// TIA Portal V19 export
FUNCTION_BLOCK "HMI_A03_FB"   // FB63, LAD
TITLE = HMI Managment
AUTHOR : Piemme
FAMILY : System
// stored: MemoryReserve 100, SetENOAutomatically false
   VAR_OUTPUT
      MB3_LpJog : Bool;
   END_VAR
   VAR
      MB3_Decoder { ExternalAccessible := 'False'; ExternalVisible := 'False'; ExternalWritable := 'False'} : "ButtonsHMIDecoder";
   END_VAR
   VAR CONSTANT
      "3002_TRASPORTO" : Int := 3002;
      "3011_FERMI_P1" : Int := 3011;
      "3012_FERMI_P1_SFALSATORE" : Int := 3012;
      "3021_FERMI_P2" : Int := 3021;
      "3022_FERMI_P2_SOLLEVATORE" : Int := 3022;
      "3031_FERMI_P3" : Int := 3031;
      "3032_SOLLEVA_RIBALTA" : Int := 3032;
      "3033_ROT_RIBALTA" : Int := 3033;
      "3034_ROT_RIBALTA_AX-POS" : Int := 3034;
      "3041_FERMI_P4" : Int := 3041;
      "3042_SPINTORE_LAT_VRT_P5" : Int := 3042;
      "3043_SPINTORE_LAT_ORZ_P5" : Int := 3043;
      "3044_SOLLEVATORI_P5" : Int := 3044;
      "3045_SPINTORE_LAT_OP" : Int := 3045;
      "3051_RIBALTATORE_OP-POS0" : Int := 3051;
      "3052_RIBALTATORE_OP-POS1" : Int := 3052;
      "3053_RIBALTATORE_OP-POS2" : Int := 3053;
      "3054_RIBALTATORE_OP-POS3" : Int := 3054;
      "4001_HU_CYTROPACK" : Int := 4001;
      "4011_SPINTORE_OP" : Int := 4011;
      "4012_SPINTORE_AX" : Int := 4012;
      "4013_SPINTORE_VRT" : Int := 4013;
      "4014_SPINTORE_ORZ" : Int := 4014;
      "4021_BORDATRICE_AX" : Int := 4021;
      "4031_RULLIERA_OP" : Int := 4031;
      "4032_RULLIERA_AX" : Int := 4032;
      "4033_BORDATRICE_REG-CASSETTA" : Int := 4033;
      "4034_BORDATRICE_PASS01" : Int := 4034;
      "4035_BORDATRICE_PASS02" : Int := 4035;
      "4036_BORDATRICE_PASS03" : Int := 4036;
      "4037_BORDATRICE_PASS04" : Int := 4037;
      "4038_BORDATRICE_REG-CASSETTA_AX-POS" : Int := 4038;
      "4041_CENTRATORI_OP" : Int := 4041;
      "4042_CENTRATORI_CENTRAGGIO" : Int := 4042;
      "4043_CENTRATORI_SOLLEVAMENTO" : Int := 4043;
      "4051_PAREGGIATORE_CODA_OP" : Int := 4051;
      "4052_PAREGGIATORE_CODA_AX" : Int := 4052;
      "4053_PAREGGIATORE_CODA_BLOCCAGGIO" : Int := 4053;
      "4054_PAREGGIATORE_CODA_BATTUTAVERTICALE" : Int := 4054;
      "4055_PAREGGIATORE_CODA_PAREGGIATORELONGIT" : Int := 4055;
      "4061_PAREGGIATORE_TESTA_OP" : Int := 4061;
      "4062_PAREGGIATORE_TESTA_AX" : Int := 4062;
      "4063_PAREGGIATORE_TESTA_BLOCCAGGIO" : Int := 4063;
      "4064_PAREGGIATORE_TESTA_SOLLEVAMENTO" : Int := 4064;
      "4065_PAREGGIATORE_TESTA_CENTRAGGIO" : Int := 4065;
      "4066_PAREGG_TESTA_AX_POS" : Int := 4066;
      "4067_PAREGG_CODA_AX_POS" : Int := 4067;
      "4070_MANIPOLATORE_OP" : Int := 4070;
      "4071_MANIPOLATORE_AX" : Int := 4071;
      "4072_MANIPOLATORE_AX-POS" : Int := 4072;
      "4073_MANIPOLATORE_MAGNETE" : Int := 4073;
      "4074_MANIPOLATORE_SOLLEVATORE" : Int := 4074;
      "4080_BORDATRICE_PASS01_LATO-OP" : Int := 4080;
      "4081_BORDATRICE_PASS01_LATO-MOT" : Int := 4081;
      "4082_BORDATRICE_PASS02_LATO-OP" : Int := 4082;
      "4083_BORDATRICE_PASS02_LATO-MOT" : Int := 4083;
      "4084_BORDATRICE_PASS03_LATO-OP" : Int := 4084;
      "4085_BORDATRICE_PASS03_LATO-MOT" : Int := 4085;
      "4086_BORDATRICE_PASS04_LATO-OP" : Int := 4086;
      "4087_BORDATRICE_PASS04_LATO-MOT" : Int := 4087;
      "4088_BORDATRICE_PASS01-COMBO_AX-POS" : Int := 4088;
      "4089_BORDATRICE_PASS02-COMBO_AX-POS" : Int := 4089;
      "4090_BORDATRICE_PASS03-COMBO_AX-POS" : Int := 4090;
      "4091_BORDATRICE_PASS04-COMBO_AX-POS" : Int := 4091;
      "4092_BORDATRICE_PASS01-LATO-OP_AX-POS" : Int := 4092;
      "4093_BORDATRICE_PASS01-LATO-MOT_AX-POS" : Int := 4093;
      "4094_BORDATRICE_PASS02-LATO-OP_AX-POS" : Int := 4094;
      "4095_BORDATRICE_PASS02-LATO-MOT_AX-POS" : Int := 4095;
      "4096_BORDATRICE_PASS03-LATO-OP_AX-POS" : Int := 4096;
      "4097_BORDATRICE_PASS03-LATO-MOT_AX-POS" : Int := 4097;
      "4098_BORDATRICE_PASS04-LATO-OP_AX-POS" : Int := 4098;
      "4099_BORDATRICE_PASS04-LATO-MOT_AX-POS" : Int := 4099;
      "5001_SPALLA_OP_POS" : Int := 5001;
      "5002_SPALLA_TESTA_AX_JOG" : Int := 5002;
      "5003_SPALLA_TESTA_AX_POS" : Int := 5003;
      "5005_SPALLA_CODA_AX" : Int := 5005;
      "5006_SPALLA_CODA_AX_POS" : Int := 5006;
      "5011_SPINTORE_OP" : Int := 5011;
      "5012_SPINTORE_VRT" : Int := 5012;
      "5013_SPINTORE_ORZ" : Int := 5013;
      "5021_TRASLAZIONE_OP_VAI_A_PRELIEVO" : Int := 5021;
      "5022_TRASLAZIONE_OP_PRELIEVO" : Int := 5022;
      "5023_TRASLAZIONE_OP_VAI_A_DEPOSITO" : Int := 5023;
      "5024_TRASLAZIONE_OP_DEPOSITO" : Int := 5024;
      "5025_TRASLAZIONE_AX_JOG" : Int := 5025;
      "5026_TRASLAZIONE_AX_POS" : Int := 5026;
      "5027_TRASLAZIONE_MANIP_SOSTEGNO" : Int := 5027;
      "5028_TRASLAZIONE_MANIP_PAREGGIATORE" : Int := 5028;
      "5029_TRASLAZIONE_SOSTEGNO_VERTICALE" : Int := 5029;
      "5031_SOLLEVAMENTO_OP" : Int := 5031;
      "5032_SOLLEVAMENTO_AX_JOG" : Int := 5032;
      "5033_SOLLEVAMENTO_AX_POS" : Int := 5033;
      "5041_PALETTIANTIRIBALTAMENTO_OP" : Int := 5041;
      "5042_PALETTIANTIRIBALTAMENTO_TESTA_POS0" : Int := 5042;
      "5043_PALETTIANTIRIBALTAMENTO_TESTA_POS1" : Int := 5043;
      "5044_PALETTIANTIRIBALTAMENTO_TESTA_POS2" : Int := 5044;
      "5046_PALETTIANTIRIBALTAMENTO_CODA_POS0" : Int := 5046;
      "5047_PALETTIANTIRIBALTAMENTO_CODA_POS1" : Int := 5047;
      "5048_PALETTIANTIRIBALTAMENTO_CODA_POS2" : Int := 5048;
      "5051_SOSTEGNO_TESTA_AX_JOG" : Int := 5051;
      "5052_SOSTEGNO_TESTA_AX_POS" : Int := 5052;
      "5053_SOSTEGNO_CODA_AX_JOG" : Int := 5053;
      "5054_SOSTEGNO_CODA_AX_POS" : Int := 5054;
      "6001_NAVETTA_OP_VAI_A_PRELIEVO" : Int := 6001;
      "6002_NAVETTA_OP_PRELIEVO" : Int := 6002;
      "6003_NAVETTA_OP_VAI_A_DEPOSITO" : Int := 6003;
      "6004_NAVETTA_OP_DEPOSITO" : Int := 6004;
      "6005_NAVETTA_AX" : Int := 6005;
      "6006_NAVETTA_PALETTI_INTERNI" : Int := 6006;
      "6007_NAVETTA_PALETTI_ESTERNI" : Int := 6007;
   END_VAR
   VAR_TEMP   // added for the SCL form of the ladder/FBD networks
      _w1 : Bool;
   END_VAR
BEGIN

REGION Network 2: <<< MB3 MANUALS OPERATIONS >>>
END_REGION

REGION Network 3 (SCL): Reset Op
   #MB3_Decoder.OpEnabled := FALSE;
   #MB3_Decoder.OpRunning := FALSE;
   #MB3_Decoder.OpDone := FALSE;
END_REGION

REGION Network 4: <<<<<<<<< A0301 STAZIONE 1 >>>>>>>>>>>>>
END_REGION

REGION Network 5: MB3 Code 3002 - Trasporto
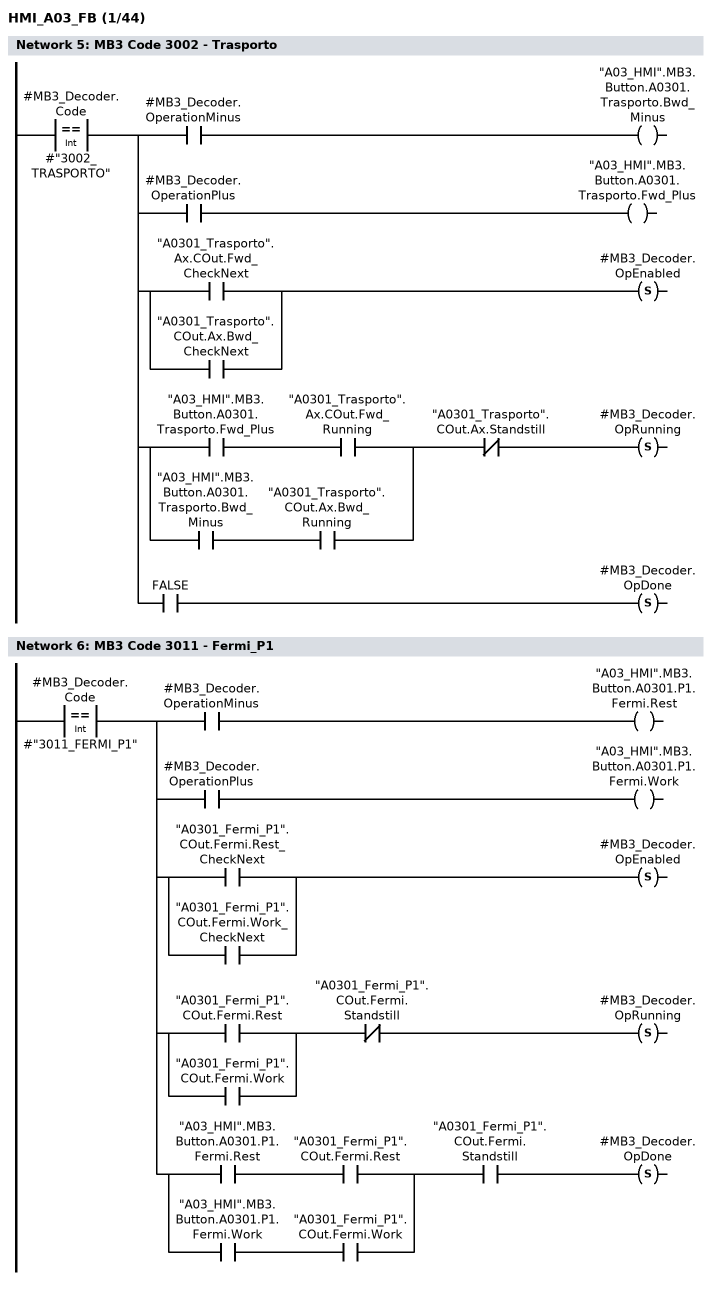
   RUNG wire#powerrail
      { S7_Templates := "SrcType := Int" } EQ_Contact(in1 := #MB3_Decoder.Code, in2 := #"3002_TRASPORTO")
      wire#w1
      Contact( #MB3_Decoder.OperationMinus )
      Coil( "A03_HMI".MB3.Button.A0301.Trasporto.Bwd_Minus )
   END_RUNG
   RUNG wire#w1
      Contact( #MB3_Decoder.OperationPlus )
      Coil( "A03_HMI".MB3.Button.A0301.Trasporto.Fwd_Plus )
   END_RUNG
   RUNG wire#w1
      Contact( "A0301_Trasporto".Ax.COut.Fwd_CheckNext )
      wire#w2
      S_Coil( #MB3_Decoder.OpEnabled )
   END_RUNG
   RUNG wire#w1
      Contact( "A0301_Trasporto".COut.Ax.Bwd_CheckNext )
   END_RUNG wire#w2
   RUNG wire#w1
      Contact( "A03_HMI".MB3.Button.A0301.Trasporto.Fwd_Plus )
      Contact( "A0301_Trasporto".Ax.COut.Fwd_Running )
      wire#w3
      I_Contact( "A0301_Trasporto".COut.Ax.Standstill )
      S_Coil( #MB3_Decoder.OpRunning )
   END_RUNG
   RUNG wire#w1
      Contact( "A03_HMI".MB3.Button.A0301.Trasporto.Bwd_Minus )
      Contact( "A0301_Trasporto".COut.Ax.Bwd_Running )
   END_RUNG wire#w3
   RUNG wire#w1
      Contact( FALSE )
      S_Coil( #MB3_Decoder.OpDone )
   END_RUNG
   // the same network as SCL:
   #_w1 := #MB3_Decoder.Code = #"3002_TRASPORTO";
   "A03_HMI".MB3.Button.A0301.Trasporto.Bwd_Minus := #_w1 AND #MB3_Decoder.OperationMinus;
   "A03_HMI".MB3.Button.A0301.Trasporto.Fwd_Plus := #_w1 AND #MB3_Decoder.OperationPlus;
   IF #_w1 AND ("A0301_Trasporto".Ax.COut.Fwd_CheckNext OR "A0301_Trasporto".COut.Ax.Bwd_CheckNext) THEN
       #MB3_Decoder.OpEnabled := TRUE;
   END_IF;
   IF #_w1 AND (("A03_HMI".MB3.Button.A0301.Trasporto.Fwd_Plus AND "A0301_Trasporto".Ax.COut.Fwd_Running) OR ("A03_HMI".MB3.Button.A0301.Trasporto.Bwd_Minus AND "A0301_Trasporto".COut.Ax.Bwd_Running)) AND NOT "A0301_Trasporto".COut.Ax.Standstill THEN
       #MB3_Decoder.OpRunning := TRUE;
   END_IF;
   IF #_w1 AND FALSE THEN #MB3_Decoder.OpDone := TRUE; END_IF;
END_REGION

REGION Network 6: MB3 Code 3011 - Fermi_P1
   RUNG wire#powerrail
      { S7_Templates := "SrcType := Int" } EQ_Contact(in1 := #MB3_Decoder.Code, in2 := #"3011_FERMI_P1")
      wire#w1
      Contact( #MB3_Decoder.OperationMinus )
      Coil( "A03_HMI".MB3.Button.A0301.P1.Fermi.Rest )
   END_RUNG
   RUNG wire#w1
      Contact( #MB3_Decoder.OperationPlus )
      Coil( "A03_HMI".MB3.Button.A0301.P1.Fermi.Work )
   END_RUNG
   RUNG wire#w1
      Contact( "A0301_Fermi_P1".COut.Fermi.Rest_CheckNext )
      wire#w2
      S_Coil( #MB3_Decoder.OpEnabled )
   END_RUNG
   RUNG wire#w1
      Contact( "A0301_Fermi_P1".COut.Fermi.Work_CheckNext )
   END_RUNG wire#w2
   RUNG wire#w1
      Contact( "A0301_Fermi_P1".COut.Fermi.Rest )
      wire#w3
      I_Contact( "A0301_Fermi_P1".COut.Fermi.Standstill )
      S_Coil( #MB3_Decoder.OpRunning )
   END_RUNG
   RUNG wire#w1
      Contact( "A0301_Fermi_P1".COut.Fermi.Work )
   END_RUNG wire#w3
   RUNG wire#w1
      Contact( "A03_HMI".MB3.Button.A0301.P1.Fermi.Rest )
      Contact( "A0301_Fermi_P1".COut.Fermi.Rest )
      wire#w4
      Contact( "A0301_Fermi_P1".COut.Fermi.Standstill )
      S_Coil( #MB3_Decoder.OpDone )
   END_RUNG
   RUNG wire#w1
      Contact( "A03_HMI".MB3.Button.A0301.P1.Fermi.Work )
      Contact( "A0301_Fermi_P1".COut.Fermi.Work )
   END_RUNG wire#w4
   // the same network as SCL:
   #_w1 := #MB3_Decoder.Code = #"3011_FERMI_P1";
   "A03_HMI".MB3.Button.A0301.P1.Fermi.Rest := #_w1 AND #MB3_Decoder.OperationMinus;
   "A03_HMI".MB3.Button.A0301.P1.Fermi.Work := #_w1 AND #MB3_Decoder.OperationPlus;
   IF #_w1 AND ("A0301_Fermi_P1".COut.Fermi.Rest_CheckNext OR "A0301_Fermi_P1".COut.Fermi.Work_CheckNext) THEN
       #MB3_Decoder.OpEnabled := TRUE;
   END_IF;
   IF #_w1 AND ("A0301_Fermi_P1".COut.Fermi.Rest OR "A0301_Fermi_P1".COut.Fermi.Work) AND NOT "A0301_Fermi_P1".COut.Fermi.Standstill THEN
       #MB3_Decoder.OpRunning := TRUE;
   END_IF;
   IF #_w1 AND (("A03_HMI".MB3.Button.A0301.P1.Fermi.Rest AND "A0301_Fermi_P1".COut.Fermi.Rest) OR ("A03_HMI".MB3.Button.A0301.P1.Fermi.Work AND "A0301_Fermi_P1".COut.Fermi.Work)) AND "A0301_Fermi_P1".COut.Fermi.Standstill THEN
       #MB3_Decoder.OpDone := TRUE;
   END_IF;
END_REGION

REGION Network 7: MB3 Code 3012 - P1 Sfalsatore
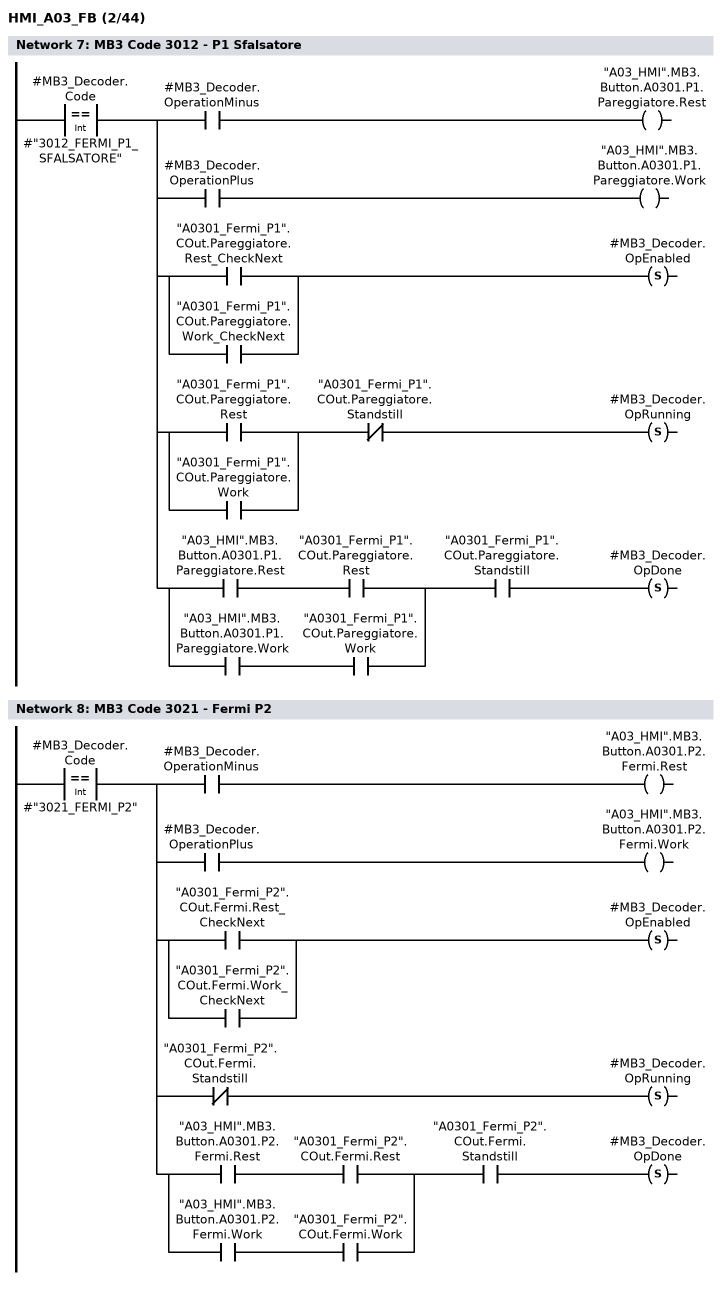
   RUNG wire#powerrail
      { S7_Templates := "SrcType := Int" } EQ_Contact(in1 := #MB3_Decoder.Code, in2 := #"3012_FERMI_P1_SFALSATORE")
      wire#w1
      Contact( #MB3_Decoder.OperationMinus )
      Coil( "A03_HMI".MB3.Button.A0301.P1.Pareggiatore.Rest )
   END_RUNG
   RUNG wire#w1
      Contact( #MB3_Decoder.OperationPlus )
      Coil( "A03_HMI".MB3.Button.A0301.P1.Pareggiatore.Work )
   END_RUNG
   RUNG wire#w1
      Contact( "A0301_Fermi_P1".COut.Pareggiatore.Rest_CheckNext )
      wire#w2
      S_Coil( #MB3_Decoder.OpEnabled )
   END_RUNG
   RUNG wire#w1
      Contact( "A0301_Fermi_P1".COut.Pareggiatore.Work_CheckNext )
   END_RUNG wire#w2
   RUNG wire#w1
      Contact( "A0301_Fermi_P1".COut.Pareggiatore.Rest )
      wire#w3
      I_Contact( "A0301_Fermi_P1".COut.Pareggiatore.Standstill )
      S_Coil( #MB3_Decoder.OpRunning )
   END_RUNG
   RUNG wire#w1
      Contact( "A0301_Fermi_P1".COut.Pareggiatore.Work )
   END_RUNG wire#w3
   RUNG wire#w1
      Contact( "A03_HMI".MB3.Button.A0301.P1.Pareggiatore.Rest )
      Contact( "A0301_Fermi_P1".COut.Pareggiatore.Rest )
      wire#w4
      Contact( "A0301_Fermi_P1".COut.Pareggiatore.Standstill )
      S_Coil( #MB3_Decoder.OpDone )
   END_RUNG
   RUNG wire#w1
      Contact( "A03_HMI".MB3.Button.A0301.P1.Pareggiatore.Work )
      Contact( "A0301_Fermi_P1".COut.Pareggiatore.Work )
   END_RUNG wire#w4
   // the same network as SCL:
   #_w1 := #MB3_Decoder.Code = #"3012_FERMI_P1_SFALSATORE";
   "A03_HMI".MB3.Button.A0301.P1.Pareggiatore.Rest := #_w1 AND #MB3_Decoder.OperationMinus;
   "A03_HMI".MB3.Button.A0301.P1.Pareggiatore.Work := #_w1 AND #MB3_Decoder.OperationPlus;
   IF #_w1 AND ("A0301_Fermi_P1".COut.Pareggiatore.Rest_CheckNext OR "A0301_Fermi_P1".COut.Pareggiatore.Work_CheckNext) THEN
       #MB3_Decoder.OpEnabled := TRUE;
   END_IF;
   IF #_w1 AND ("A0301_Fermi_P1".COut.Pareggiatore.Rest OR "A0301_Fermi_P1".COut.Pareggiatore.Work) AND NOT "A0301_Fermi_P1".COut.Pareggiatore.Standstill THEN
       #MB3_Decoder.OpRunning := TRUE;
   END_IF;
   IF #_w1 AND (("A03_HMI".MB3.Button.A0301.P1.Pareggiatore.Rest AND "A0301_Fermi_P1".COut.Pareggiatore.Rest) OR ("A03_HMI".MB3.Button.A0301.P1.Pareggiatore.Work AND "A0301_Fermi_P1".COut.Pareggiatore.Work)) AND "A0301_Fermi_P1".COut.Pareggiatore.Standstill THEN
       #MB3_Decoder.OpDone := TRUE;
   END_IF;
END_REGION

REGION Network 8: MB3 Code 3021 - Fermi P2
   RUNG wire#powerrail
      { S7_Templates := "SrcType := Int" } EQ_Contact(in1 := #MB3_Decoder.Code, in2 := #"3021_FERMI_P2")
      wire#w1
      Contact( #MB3_Decoder.OperationMinus )
      Coil( "A03_HMI".MB3.Button.A0301.P2.Fermi.Rest )
   END_RUNG
   RUNG wire#w1
      Contact( #MB3_Decoder.OperationPlus )
      Coil( "A03_HMI".MB3.Button.A0301.P2.Fermi.Work )
   END_RUNG
   RUNG wire#w1
      Contact( "A0301_Fermi_P2".COut.Fermi.Rest_CheckNext )
      wire#w2
      S_Coil( #MB3_Decoder.OpEnabled )
   END_RUNG
   RUNG wire#w1
      Contact( "A0301_Fermi_P2".COut.Fermi.Work_CheckNext )
   END_RUNG wire#w2
   RUNG wire#w1
      I_Contact( "A0301_Fermi_P2".COut.Fermi.Standstill )
      S_Coil( #MB3_Decoder.OpRunning )
   END_RUNG
   RUNG wire#w1
      Contact( "A03_HMI".MB3.Button.A0301.P2.Fermi.Rest )
      Contact( "A0301_Fermi_P2".COut.Fermi.Rest )
      wire#w3
      Contact( "A0301_Fermi_P2".COut.Fermi.Standstill )
      S_Coil( #MB3_Decoder.OpDone )
   END_RUNG
   RUNG wire#w1
      Contact( "A03_HMI".MB3.Button.A0301.P2.Fermi.Work )
      Contact( "A0301_Fermi_P2".COut.Fermi.Work )
   END_RUNG wire#w3
   // the same network as SCL:
   #_w1 := #MB3_Decoder.Code = #"3021_FERMI_P2";
   "A03_HMI".MB3.Button.A0301.P2.Fermi.Rest := #_w1 AND #MB3_Decoder.OperationMinus;
   "A03_HMI".MB3.Button.A0301.P2.Fermi.Work := #_w1 AND #MB3_Decoder.OperationPlus;
   IF #_w1 AND ("A0301_Fermi_P2".COut.Fermi.Rest_CheckNext OR "A0301_Fermi_P2".COut.Fermi.Work_CheckNext) THEN
       #MB3_Decoder.OpEnabled := TRUE;
   END_IF;
   IF #_w1 AND NOT "A0301_Fermi_P2".COut.Fermi.Standstill THEN #MB3_Decoder.OpRunning := TRUE; END_IF;
   IF #_w1 AND (("A03_HMI".MB3.Button.A0301.P2.Fermi.Rest AND "A0301_Fermi_P2".COut.Fermi.Rest) OR ("A03_HMI".MB3.Button.A0301.P2.Fermi.Work AND "A0301_Fermi_P2".COut.Fermi.Work)) AND "A0301_Fermi_P2".COut.Fermi.Standstill THEN
       #MB3_Decoder.OpDone := TRUE;
   END_IF;
END_REGION

REGION Network 9: MB3 Code 3022 - P2 - Sollevatore
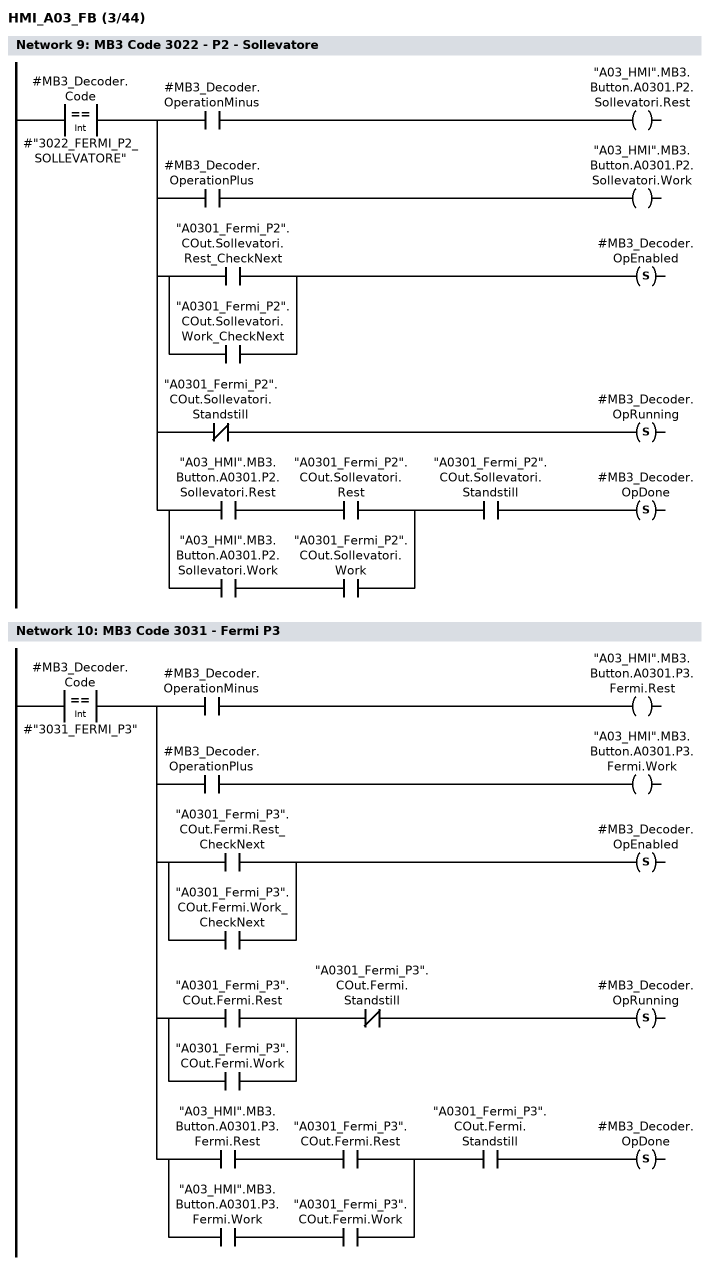
   RUNG wire#powerrail
      { S7_Templates := "SrcType := Int" } EQ_Contact(in1 := #MB3_Decoder.Code, in2 := #"3022_FERMI_P2_SOLLEVATORE")
      wire#w1
      Contact( #MB3_Decoder.OperationMinus )
      Coil( "A03_HMI".MB3.Button.A0301.P2.Sollevatori.Rest )
   END_RUNG
   RUNG wire#w1
      Contact( #MB3_Decoder.OperationPlus )
      Coil( "A03_HMI".MB3.Button.A0301.P2.Sollevatori.Work )
   END_RUNG
   RUNG wire#w1
      Contact( "A0301_Fermi_P2".COut.Sollevatori.Rest_CheckNext )
      wire#w2
      S_Coil( #MB3_Decoder.OpEnabled )
   END_RUNG
   RUNG wire#w1
      Contact( "A0301_Fermi_P2".COut.Sollevatori.Work_CheckNext )
   END_RUNG wire#w2
   RUNG wire#w1
      I_Contact( "A0301_Fermi_P2".COut.Sollevatori.Standstill )
      S_Coil( #MB3_Decoder.OpRunning )
   END_RUNG
   RUNG wire#w1
      Contact( "A03_HMI".MB3.Button.A0301.P2.Sollevatori.Rest )
      Contact( "A0301_Fermi_P2".COut.Sollevatori.Rest )
      wire#w3
      Contact( "A0301_Fermi_P2".COut.Sollevatori.Standstill )
      S_Coil( #MB3_Decoder.OpDone )
   END_RUNG
   RUNG wire#w1
      Contact( "A03_HMI".MB3.Button.A0301.P2.Sollevatori.Work )
      Contact( "A0301_Fermi_P2".COut.Sollevatori.Work )
   END_RUNG wire#w3
   // the same network as SCL:
   #_w1 := #MB3_Decoder.Code = #"3022_FERMI_P2_SOLLEVATORE";
   "A03_HMI".MB3.Button.A0301.P2.Sollevatori.Rest := #_w1 AND #MB3_Decoder.OperationMinus;
   "A03_HMI".MB3.Button.A0301.P2.Sollevatori.Work := #_w1 AND #MB3_Decoder.OperationPlus;
   IF #_w1 AND ("A0301_Fermi_P2".COut.Sollevatori.Rest_CheckNext OR "A0301_Fermi_P2".COut.Sollevatori.Work_CheckNext) THEN
       #MB3_Decoder.OpEnabled := TRUE;
   END_IF;
   IF #_w1 AND NOT "A0301_Fermi_P2".COut.Sollevatori.Standstill THEN #MB3_Decoder.OpRunning := TRUE; END_IF;
   IF #_w1 AND (("A03_HMI".MB3.Button.A0301.P2.Sollevatori.Rest AND "A0301_Fermi_P2".COut.Sollevatori.Rest) OR ("A03_HMI".MB3.Button.A0301.P2.Sollevatori.Work AND "A0301_Fermi_P2".COut.Sollevatori.Work)) AND "A0301_Fermi_P2".COut.Sollevatori.Standstill THEN
       #MB3_Decoder.OpDone := TRUE;
   END_IF;
END_REGION

REGION Network 10: MB3 Code 3031 - Fermi P3
   RUNG wire#powerrail
      { S7_Templates := "SrcType := Int" } EQ_Contact(in1 := #MB3_Decoder.Code, in2 := #"3031_FERMI_P3")
      wire#w1
      Contact( #MB3_Decoder.OperationMinus )
      Coil( "A03_HMI".MB3.Button.A0301.P3.Fermi.Rest )
   END_RUNG
   RUNG wire#w1
      Contact( #MB3_Decoder.OperationPlus )
      Coil( "A03_HMI".MB3.Button.A0301.P3.Fermi.Work )
   END_RUNG
   RUNG wire#w1
      Contact( "A0301_Fermi_P3".COut.Fermi.Rest_CheckNext )
      wire#w2
      S_Coil( #MB3_Decoder.OpEnabled )
   END_RUNG
   RUNG wire#w1
      Contact( "A0301_Fermi_P3".COut.Fermi.Work_CheckNext )
   END_RUNG wire#w2
   RUNG wire#w1
      Contact( "A0301_Fermi_P3".COut.Fermi.Rest )
      wire#w3
      I_Contact( "A0301_Fermi_P3".COut.Fermi.Standstill )
      S_Coil( #MB3_Decoder.OpRunning )
   END_RUNG
   RUNG wire#w1
      Contact( "A0301_Fermi_P3".COut.Fermi.Work )
   END_RUNG wire#w3
   RUNG wire#w1
      Contact( "A03_HMI".MB3.Button.A0301.P3.Fermi.Rest )
      Contact( "A0301_Fermi_P3".COut.Fermi.Rest )
      wire#w4
      Contact( "A0301_Fermi_P3".COut.Fermi.Standstill )
      S_Coil( #MB3_Decoder.OpDone )
   END_RUNG
   RUNG wire#w1
      Contact( "A03_HMI".MB3.Button.A0301.P3.Fermi.Work )
      Contact( "A0301_Fermi_P3".COut.Fermi.Work )
   END_RUNG wire#w4
   // the same network as SCL:
   #_w1 := #MB3_Decoder.Code = #"3031_FERMI_P3";
   "A03_HMI".MB3.Button.A0301.P3.Fermi.Rest := #_w1 AND #MB3_Decoder.OperationMinus;
   "A03_HMI".MB3.Button.A0301.P3.Fermi.Work := #_w1 AND #MB3_Decoder.OperationPlus;
   IF #_w1 AND ("A0301_Fermi_P3".COut.Fermi.Rest_CheckNext OR "A0301_Fermi_P3".COut.Fermi.Work_CheckNext) THEN
       #MB3_Decoder.OpEnabled := TRUE;
   END_IF;
   IF #_w1 AND ("A0301_Fermi_P3".COut.Fermi.Rest OR "A0301_Fermi_P3".COut.Fermi.Work) AND NOT "A0301_Fermi_P3".COut.Fermi.Standstill THEN
       #MB3_Decoder.OpRunning := TRUE;
   END_IF;
   IF #_w1 AND (("A03_HMI".MB3.Button.A0301.P3.Fermi.Rest AND "A0301_Fermi_P3".COut.Fermi.Rest) OR ("A03_HMI".MB3.Button.A0301.P3.Fermi.Work AND "A0301_Fermi_P3".COut.Fermi.Work)) AND "A0301_Fermi_P3".COut.Fermi.Standstill THEN
       #MB3_Decoder.OpDone := TRUE;
   END_IF;
END_REGION

REGION Network 11: MB3 Code 3032 - Solleva Ribalta
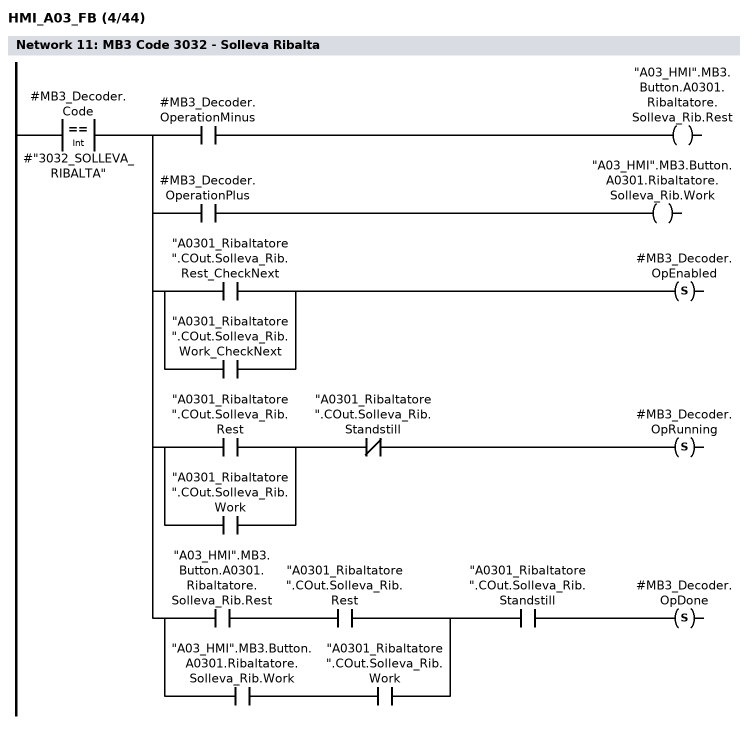
   RUNG wire#powerrail
      { S7_Templates := "SrcType := Int" } EQ_Contact(in1 := #MB3_Decoder.Code, in2 := #"3032_SOLLEVA_RIBALTA")
      wire#w1
      Contact( #MB3_Decoder.OperationMinus )
      Coil( "A03_HMI".MB3.Button.A0301.Ribaltatore.Solleva_Rib.Rest )
   END_RUNG
   RUNG wire#w1
      Contact( #MB3_Decoder.OperationPlus )
      Coil( "A03_HMI".MB3.Button.A0301.Ribaltatore.Solleva_Rib.Work )
   END_RUNG
   RUNG wire#w1
      Contact( "A0301_Ribaltatore".COut.Solleva_Rib.Rest_CheckNext )
      wire#w2
      S_Coil( #MB3_Decoder.OpEnabled )
   END_RUNG
   RUNG wire#w1
      Contact( "A0301_Ribaltatore".COut.Solleva_Rib.Work_CheckNext )
   END_RUNG wire#w2
   RUNG wire#w1
      Contact( "A0301_Ribaltatore".COut.Solleva_Rib.Rest )
      wire#w3
      I_Contact( "A0301_Ribaltatore".COut.Solleva_Rib.Standstill )
      S_Coil( #MB3_Decoder.OpRunning )
   END_RUNG
   RUNG wire#w1
      Contact( "A0301_Ribaltatore".COut.Solleva_Rib.Work )
   END_RUNG wire#w3
   RUNG wire#w1
      Contact( "A03_HMI".MB3.Button.A0301.Ribaltatore.Solleva_Rib.Rest )
      Contact( "A0301_Ribaltatore".COut.Solleva_Rib.Rest )
      wire#w4
      Contact( "A0301_Ribaltatore".COut.Solleva_Rib.Standstill )
      S_Coil( #MB3_Decoder.OpDone )
   END_RUNG
   RUNG wire#w1
      Contact( "A03_HMI".MB3.Button.A0301.Ribaltatore.Solleva_Rib.Work )
      Contact( "A0301_Ribaltatore".COut.Solleva_Rib.Work )
   END_RUNG wire#w4
   // the same network as SCL:
   #_w1 := #MB3_Decoder.Code = #"3032_SOLLEVA_RIBALTA";
   "A03_HMI".MB3.Button.A0301.Ribaltatore.Solleva_Rib.Rest := #_w1 AND #MB3_Decoder.OperationMinus;
   "A03_HMI".MB3.Button.A0301.Ribaltatore.Solleva_Rib.Work := #_w1 AND #MB3_Decoder.OperationPlus;
   IF #_w1 AND ("A0301_Ribaltatore".COut.Solleva_Rib.Rest_CheckNext OR "A0301_Ribaltatore".COut.Solleva_Rib.Work_CheckNext) THEN
       #MB3_Decoder.OpEnabled := TRUE;
   END_IF;
   IF #_w1 AND ("A0301_Ribaltatore".COut.Solleva_Rib.Rest OR "A0301_Ribaltatore".COut.Solleva_Rib.Work) AND NOT "A0301_Ribaltatore".COut.Solleva_Rib.Standstill THEN
       #MB3_Decoder.OpRunning := TRUE;
   END_IF;
   IF #_w1 AND (("A03_HMI".MB3.Button.A0301.Ribaltatore.Solleva_Rib.Rest AND "A0301_Ribaltatore".COut.Solleva_Rib.Rest) OR ("A03_HMI".MB3.Button.A0301.Ribaltatore.Solleva_Rib.Work AND "A0301_Ribaltatore".COut.Solleva_Rib.Work)) AND "A0301_Ribaltatore".COut.Solleva_Rib.Standstill THEN
       #MB3_Decoder.OpDone := TRUE;
   END_IF;
END_REGION

REGION Network 12: MB3 Code 3033 - Rotazione Ribalta
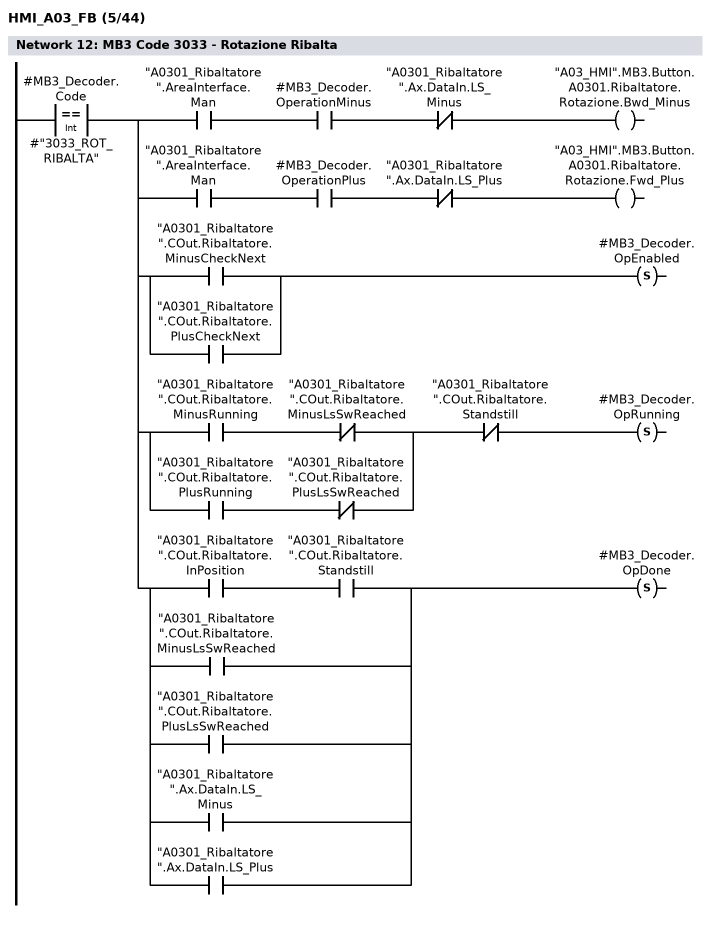
   RUNG wire#powerrail
      { S7_Templates := "SrcType := Int" } EQ_Contact(in1 := #MB3_Decoder.Code, in2 := #"3033_ROT_RIBALTA")
      wire#w1
      Contact( "A0301_Ribaltatore".AreaInterface.Man )
      Contact( #MB3_Decoder.OperationMinus )
      I_Contact( "A0301_Ribaltatore".Ax.DataIn.LS_Minus )
      Coil( "A03_HMI".MB3.Button.A0301.Ribaltatore.Rotazione.Bwd_Minus )
   END_RUNG
   RUNG wire#w1
      Contact( "A0301_Ribaltatore".AreaInterface.Man )
      Contact( #MB3_Decoder.OperationPlus )
      I_Contact( "A0301_Ribaltatore".Ax.DataIn.LS_Plus )
      Coil( "A03_HMI".MB3.Button.A0301.Ribaltatore.Rotazione.Fwd_Plus )
   END_RUNG
   RUNG wire#w1
      Contact( "A0301_Ribaltatore".COut.Ribaltatore.MinusCheckNext )
      wire#w2
      S_Coil( #MB3_Decoder.OpEnabled )
   END_RUNG
   RUNG wire#w1
      Contact( "A0301_Ribaltatore".COut.Ribaltatore.PlusCheckNext )
   END_RUNG wire#w2
   RUNG wire#w1
      Contact( "A0301_Ribaltatore".COut.Ribaltatore.MinusRunning )
      I_Contact( "A0301_Ribaltatore".COut.Ribaltatore.MinusLsSwReached )
      wire#w3
      I_Contact( "A0301_Ribaltatore".COut.Ribaltatore.Standstill )
      S_Coil( #MB3_Decoder.OpRunning )
   END_RUNG
   RUNG wire#w1
      Contact( "A0301_Ribaltatore".COut.Ribaltatore.PlusRunning )
      I_Contact( "A0301_Ribaltatore".COut.Ribaltatore.PlusLsSwReached )
   END_RUNG wire#w3
   RUNG wire#w1
      Contact( "A0301_Ribaltatore".COut.Ribaltatore.InPosition )
      Contact( "A0301_Ribaltatore".COut.Ribaltatore.Standstill )
      wire#w4
      S_Coil( #MB3_Decoder.OpDone )
   END_RUNG
   RUNG wire#w1
      Contact( "A0301_Ribaltatore".COut.Ribaltatore.MinusLsSwReached )
   END_RUNG wire#w4
   RUNG wire#w1
      Contact( "A0301_Ribaltatore".COut.Ribaltatore.PlusLsSwReached )
   END_RUNG wire#w4
   RUNG wire#w1
      Contact( "A0301_Ribaltatore".Ax.DataIn.LS_Minus )
   END_RUNG wire#w4
   RUNG wire#w1
      Contact( "A0301_Ribaltatore".Ax.DataIn.LS_Plus )
   END_RUNG wire#w4
   // the same network as SCL:
   #_w1 := #MB3_Decoder.Code = #"3033_ROT_RIBALTA";
   "A03_HMI".MB3.Button.A0301.Ribaltatore.Rotazione.Bwd_Minus := #_w1 AND "A0301_Ribaltatore".AreaInterface.Man AND #MB3_Decoder.OperationMinus AND NOT "A0301_Ribaltatore".Ax.DataIn.LS_Minus;
   "A03_HMI".MB3.Button.A0301.Ribaltatore.Rotazione.Fwd_Plus := #_w1 AND "A0301_Ribaltatore".AreaInterface.Man AND #MB3_Decoder.OperationPlus AND NOT "A0301_Ribaltatore".Ax.DataIn.LS_Plus;
   IF #_w1 AND ("A0301_Ribaltatore".COut.Ribaltatore.MinusCheckNext OR "A0301_Ribaltatore".COut.Ribaltatore.PlusCheckNext) THEN
       #MB3_Decoder.OpEnabled := TRUE;
   END_IF;
   IF #_w1 AND (("A0301_Ribaltatore".COut.Ribaltatore.MinusRunning AND NOT "A0301_Ribaltatore".COut.Ribaltatore.MinusLsSwReached) OR ("A0301_Ribaltatore".COut.Ribaltatore.PlusRunning AND NOT "A0301_Ribaltatore".COut.Ribaltatore.PlusLsSwReached)) AND NOT "A0301_Ribaltatore".COut.Ribaltatore.Standstill THEN
       #MB3_Decoder.OpRunning := TRUE;
   END_IF;
   IF #_w1 AND (("A0301_Ribaltatore".COut.Ribaltatore.InPosition AND "A0301_Ribaltatore".COut.Ribaltatore.Standstill) OR "A0301_Ribaltatore".COut.Ribaltatore.MinusLsSwReached OR "A0301_Ribaltatore".COut.Ribaltatore.PlusLsSwReached OR "A0301_Ribaltatore".Ax.DataIn.LS_Minus OR "A0301_Ribaltatore".Ax.DataIn.LS_Plus) THEN
       #MB3_Decoder.OpDone := TRUE;
   END_IF;
END_REGION

REGION Network 13: MB3 Code 3034 - Rotazione Ribalta -AX_POS
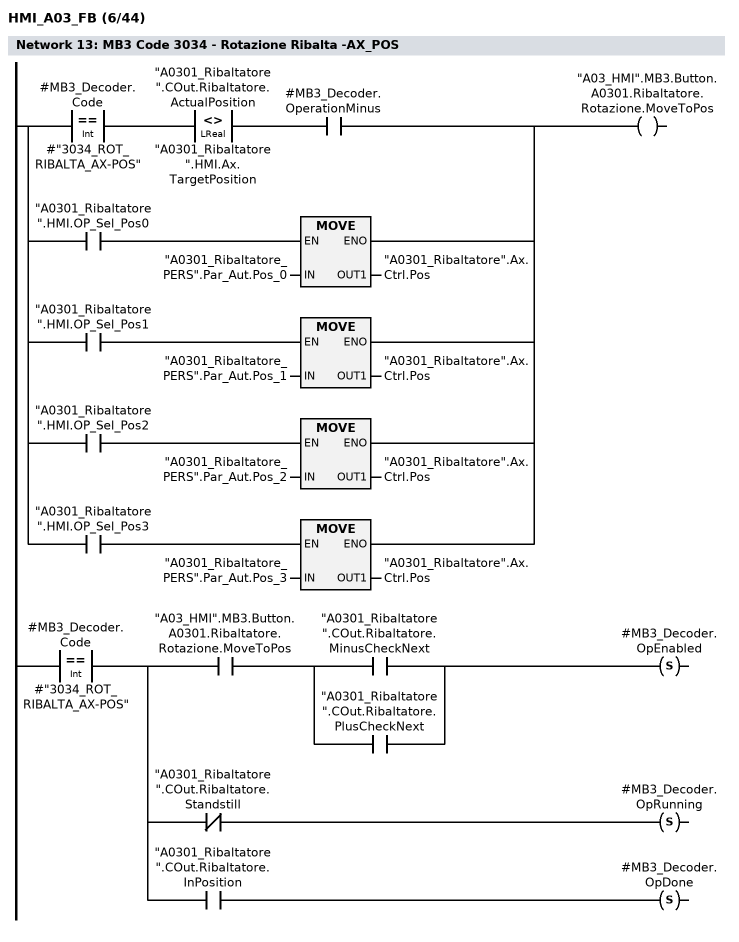
   RUNG wire#powerrail
      { S7_Templates := "SrcType := Int" } EQ_Contact(in1 := #MB3_Decoder.Code, in2 := #"3034_ROT_RIBALTA_AX-POS")
      { S7_Templates := "SrcType := LReal" } NE_Contact(in1 := "A0301_Ribaltatore".COut.Ribaltatore.ActualPosition, in2 := "A0301_Ribaltatore".HMI.Ax.TargetPosition)
      Contact( #MB3_Decoder.OperationMinus )
      wire#w1
      Coil( "A03_HMI".MB3.Button.A0301.Ribaltatore.Rotazione.MoveToPos )
   END_RUNG
   RUNG wire#powerrail
      Contact( "A0301_Ribaltatore".HMI.OP_Sel_Pos0 )
      Move(in := "A0301_Ribaltatore_PERS".Par_Aut.Pos_0, out1 => "A0301_Ribaltatore".Ax.Ctrl.Pos)
   END_RUNG wire#w1
   RUNG wire#powerrail
      Contact( "A0301_Ribaltatore".HMI.OP_Sel_Pos1 )
      Move(in := "A0301_Ribaltatore_PERS".Par_Aut.Pos_1, out1 => "A0301_Ribaltatore".Ax.Ctrl.Pos)
   END_RUNG wire#w1
   RUNG wire#powerrail
      Contact( "A0301_Ribaltatore".HMI.OP_Sel_Pos2 )
      Move(in := "A0301_Ribaltatore_PERS".Par_Aut.Pos_2, out1 => "A0301_Ribaltatore".Ax.Ctrl.Pos)
   END_RUNG wire#w1
   RUNG wire#powerrail
      Contact( "A0301_Ribaltatore".HMI.OP_Sel_Pos3 )
      Move(in := "A0301_Ribaltatore_PERS".Par_Aut.Pos_3, out1 => "A0301_Ribaltatore".Ax.Ctrl.Pos)
   END_RUNG wire#w1
   RUNG wire#powerrail
      { S7_Templates := "SrcType := Int" } EQ_Contact(in1 := #MB3_Decoder.Code, in2 := #"3034_ROT_RIBALTA_AX-POS")
      wire#w2
      Contact( "A03_HMI".MB3.Button.A0301.Ribaltatore.Rotazione.MoveToPos )
      wire#w3
      Contact( "A0301_Ribaltatore".COut.Ribaltatore.MinusCheckNext )
      wire#w4
      S_Coil( #MB3_Decoder.OpEnabled )
   END_RUNG
   RUNG wire#w3
      Contact( "A0301_Ribaltatore".COut.Ribaltatore.PlusCheckNext )
   END_RUNG wire#w4
   RUNG wire#w2
      I_Contact( "A0301_Ribaltatore".COut.Ribaltatore.Standstill )
      S_Coil( #MB3_Decoder.OpRunning )
   END_RUNG
   RUNG wire#w2
      Contact( "A0301_Ribaltatore".COut.Ribaltatore.InPosition )
      S_Coil( #MB3_Decoder.OpDone )
   END_RUNG
   // the same network as SCL:
   IF "A0301_Ribaltatore".HMI.OP_Sel_Pos0 THEN
       "A0301_Ribaltatore".Ax.Ctrl.Pos := "A0301_Ribaltatore_PERS".Par_Aut.Pos_0;
   END_IF;
   IF "A0301_Ribaltatore".HMI.OP_Sel_Pos1 THEN
       "A0301_Ribaltatore".Ax.Ctrl.Pos := "A0301_Ribaltatore_PERS".Par_Aut.Pos_1;
   END_IF;
   IF "A0301_Ribaltatore".HMI.OP_Sel_Pos2 THEN
       "A0301_Ribaltatore".Ax.Ctrl.Pos := "A0301_Ribaltatore_PERS".Par_Aut.Pos_2;
   END_IF;
   IF "A0301_Ribaltatore".HMI.OP_Sel_Pos3 THEN
       "A0301_Ribaltatore".Ax.Ctrl.Pos := "A0301_Ribaltatore_PERS".Par_Aut.Pos_3;
   END_IF;
   "A03_HMI".MB3.Button.A0301.Ribaltatore.Rotazione.MoveToPos := ((#MB3_Decoder.Code = #"3034_ROT_RIBALTA_AX-POS") AND ("A0301_Ribaltatore".COut.Ribaltatore.ActualPosition <> "A0301_Ribaltatore".HMI.Ax.TargetPosition) AND #MB3_Decoder.OperationMinus) OR "A0301_Ribaltatore".HMI.OP_Sel_Pos0 OR "A0301_Ribaltatore".HMI.OP_Sel_Pos1 OR "A0301_Ribaltatore".HMI.OP_Sel_Pos2 OR "A0301_Ribaltatore".HMI.OP_Sel_Pos3;
   #_w1 := #MB3_Decoder.Code = #"3034_ROT_RIBALTA_AX-POS";
   IF #_w1 AND "A03_HMI".MB3.Button.A0301.Ribaltatore.Rotazione.MoveToPos AND ("A0301_Ribaltatore".COut.Ribaltatore.MinusCheckNext OR "A0301_Ribaltatore".COut.Ribaltatore.PlusCheckNext) THEN
       #MB3_Decoder.OpEnabled := TRUE;
   END_IF;
   IF #_w1 AND NOT "A0301_Ribaltatore".COut.Ribaltatore.Standstill THEN
       #MB3_Decoder.OpRunning := TRUE;
   END_IF;
   IF #_w1 AND "A0301_Ribaltatore".COut.Ribaltatore.InPosition THEN #MB3_Decoder.OpDone := TRUE; END_IF;
END_REGION

REGION Network 14: MB3 Code 6008 - Rotazione Ribalta - OP POS0
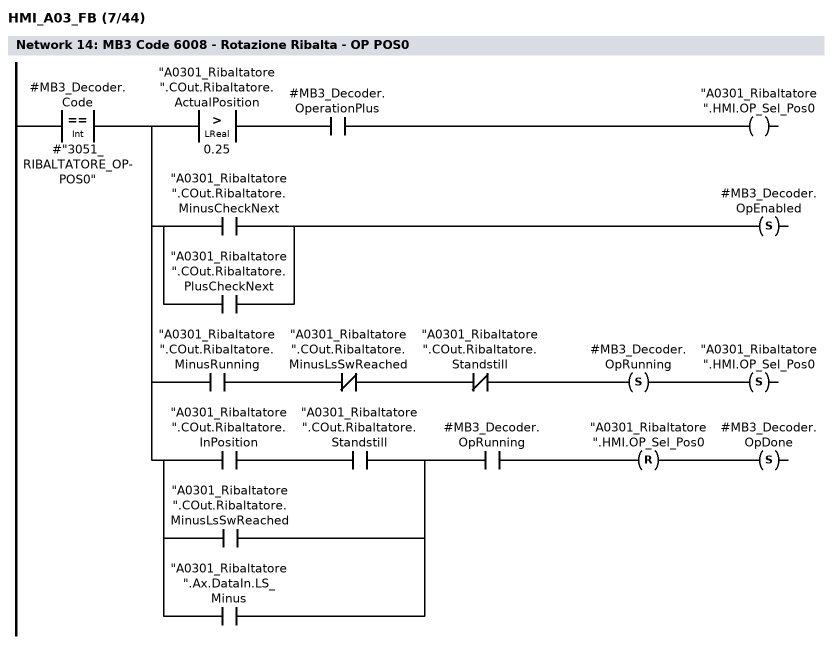
   RUNG wire#powerrail
      { S7_Templates := "SrcType := Int" } EQ_Contact(in1 := #MB3_Decoder.Code, in2 := #"3051_RIBALTATORE_OP-POS0")
      wire#w1
      { S7_Templates := "SrcType := LReal" } GT_Contact(in1 := "A0301_Ribaltatore".COut.Ribaltatore.ActualPosition, in2 := 0.25)
      Contact( #MB3_Decoder.OperationPlus )
      Coil( "A0301_Ribaltatore".HMI.OP_Sel_Pos0 )
   END_RUNG
   RUNG wire#w1
      Contact( "A0301_Ribaltatore".COut.Ribaltatore.MinusCheckNext )
      wire#w2
      S_Coil( #MB3_Decoder.OpEnabled )
   END_RUNG
   RUNG wire#w1
      Contact( "A0301_Ribaltatore".COut.Ribaltatore.PlusCheckNext )
   END_RUNG wire#w2
   RUNG wire#w1
      Contact( "A0301_Ribaltatore".COut.Ribaltatore.MinusRunning )
      I_Contact( "A0301_Ribaltatore".COut.Ribaltatore.MinusLsSwReached )
      I_Contact( "A0301_Ribaltatore".COut.Ribaltatore.Standstill )
      S_Coil( #MB3_Decoder.OpRunning )
      S_Coil( "A0301_Ribaltatore".HMI.OP_Sel_Pos0 )
   END_RUNG
   RUNG wire#w1
      Contact( "A0301_Ribaltatore".COut.Ribaltatore.InPosition )
      Contact( "A0301_Ribaltatore".COut.Ribaltatore.Standstill )
      wire#w3
      Contact( #MB3_Decoder.OpRunning )
      R_Coil( "A0301_Ribaltatore".HMI.OP_Sel_Pos0 )
      S_Coil( #MB3_Decoder.OpDone )
   END_RUNG
   RUNG wire#w1
      Contact( "A0301_Ribaltatore".COut.Ribaltatore.MinusLsSwReached )
   END_RUNG wire#w3
   RUNG wire#w1
      Contact( "A0301_Ribaltatore".Ax.DataIn.LS_Minus )
   END_RUNG wire#w3
   // the same network as SCL:
   #_w1 := #MB3_Decoder.Code = #"3051_RIBALTATORE_OP-POS0";
   "A0301_Ribaltatore".HMI.OP_Sel_Pos0 := #_w1 AND ("A0301_Ribaltatore".COut.Ribaltatore.ActualPosition > 0.25) AND #MB3_Decoder.OperationPlus;
   IF #_w1 AND ("A0301_Ribaltatore".COut.Ribaltatore.MinusCheckNext OR "A0301_Ribaltatore".COut.Ribaltatore.PlusCheckNext) THEN
       #MB3_Decoder.OpEnabled := TRUE;
   END_IF;
   IF #_w1 AND "A0301_Ribaltatore".COut.Ribaltatore.MinusRunning AND NOT "A0301_Ribaltatore".COut.Ribaltatore.MinusLsSwReached AND NOT "A0301_Ribaltatore".COut.Ribaltatore.Standstill THEN
       #MB3_Decoder.OpRunning := TRUE;
       "A0301_Ribaltatore".HMI.OP_Sel_Pos0 := TRUE;
   END_IF;
   IF #_w1 AND (("A0301_Ribaltatore".COut.Ribaltatore.InPosition AND "A0301_Ribaltatore".COut.Ribaltatore.Standstill) OR "A0301_Ribaltatore".COut.Ribaltatore.MinusLsSwReached OR "A0301_Ribaltatore".Ax.DataIn.LS_Minus) AND #MB3_Decoder.OpRunning THEN
       "A0301_Ribaltatore".HMI.OP_Sel_Pos0 := FALSE;
       #MB3_Decoder.OpDone := TRUE;
   END_IF;
END_REGION

REGION Network 15: MB3 Code 6009 - Rotazione Ribalta - OP POS1
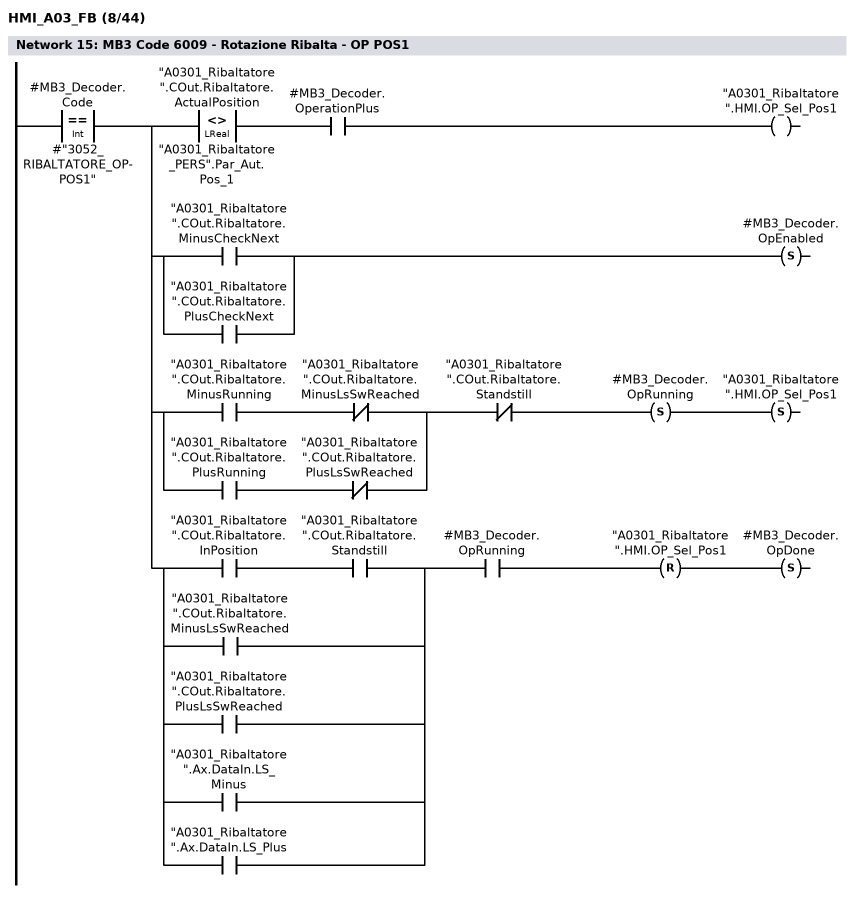
   RUNG wire#powerrail
      { S7_Templates := "SrcType := Int" } EQ_Contact(in1 := #MB3_Decoder.Code, in2 := #"3052_RIBALTATORE_OP-POS1")
      wire#w1
      { S7_Templates := "SrcType := LReal" } NE_Contact(in1 := "A0301_Ribaltatore".COut.Ribaltatore.ActualPosition, in2 := "A0301_Ribaltatore_PERS".Par_Aut.Pos_1)
      Contact( #MB3_Decoder.OperationPlus )
      Coil( "A0301_Ribaltatore".HMI.OP_Sel_Pos1 )
   END_RUNG
   RUNG wire#w1
      Contact( "A0301_Ribaltatore".COut.Ribaltatore.MinusCheckNext )
      wire#w2
      S_Coil( #MB3_Decoder.OpEnabled )
   END_RUNG
   RUNG wire#w1
      Contact( "A0301_Ribaltatore".COut.Ribaltatore.PlusCheckNext )
   END_RUNG wire#w2
   RUNG wire#w1
      Contact( "A0301_Ribaltatore".COut.Ribaltatore.MinusRunning )
      I_Contact( "A0301_Ribaltatore".COut.Ribaltatore.MinusLsSwReached )
      wire#w3
      I_Contact( "A0301_Ribaltatore".COut.Ribaltatore.Standstill )
      S_Coil( #MB3_Decoder.OpRunning )
      S_Coil( "A0301_Ribaltatore".HMI.OP_Sel_Pos1 )
   END_RUNG
   RUNG wire#w1
      Contact( "A0301_Ribaltatore".COut.Ribaltatore.PlusRunning )
      I_Contact( "A0301_Ribaltatore".COut.Ribaltatore.PlusLsSwReached )
   END_RUNG wire#w3
   RUNG wire#w1
      Contact( "A0301_Ribaltatore".COut.Ribaltatore.InPosition )
      Contact( "A0301_Ribaltatore".COut.Ribaltatore.Standstill )
      wire#w4
      Contact( #MB3_Decoder.OpRunning )
      R_Coil( "A0301_Ribaltatore".HMI.OP_Sel_Pos1 )
      S_Coil( #MB3_Decoder.OpDone )
   END_RUNG
   RUNG wire#w1
      Contact( "A0301_Ribaltatore".COut.Ribaltatore.MinusLsSwReached )
   END_RUNG wire#w4
   RUNG wire#w1
      Contact( "A0301_Ribaltatore".COut.Ribaltatore.PlusLsSwReached )
   END_RUNG wire#w4
   RUNG wire#w1
      Contact( "A0301_Ribaltatore".Ax.DataIn.LS_Minus )
   END_RUNG wire#w4
   RUNG wire#w1
      Contact( "A0301_Ribaltatore".Ax.DataIn.LS_Plus )
   END_RUNG wire#w4
   // the same network as SCL:
   #_w1 := #MB3_Decoder.Code = #"3052_RIBALTATORE_OP-POS1";
   "A0301_Ribaltatore".HMI.OP_Sel_Pos1 := #_w1 AND ("A0301_Ribaltatore".COut.Ribaltatore.ActualPosition <> "A0301_Ribaltatore_PERS".Par_Aut.Pos_1) AND #MB3_Decoder.OperationPlus;
   IF #_w1 AND ("A0301_Ribaltatore".COut.Ribaltatore.MinusCheckNext OR "A0301_Ribaltatore".COut.Ribaltatore.PlusCheckNext) THEN
       #MB3_Decoder.OpEnabled := TRUE;
   END_IF;
   IF #_w1 AND (("A0301_Ribaltatore".COut.Ribaltatore.MinusRunning AND NOT "A0301_Ribaltatore".COut.Ribaltatore.MinusLsSwReached) OR ("A0301_Ribaltatore".COut.Ribaltatore.PlusRunning AND NOT "A0301_Ribaltatore".COut.Ribaltatore.PlusLsSwReached)) AND NOT "A0301_Ribaltatore".COut.Ribaltatore.Standstill THEN
       #MB3_Decoder.OpRunning := TRUE;
       "A0301_Ribaltatore".HMI.OP_Sel_Pos1 := TRUE;
   END_IF;
   IF #_w1 AND (("A0301_Ribaltatore".COut.Ribaltatore.InPosition AND "A0301_Ribaltatore".COut.Ribaltatore.Standstill) OR "A0301_Ribaltatore".COut.Ribaltatore.MinusLsSwReached OR "A0301_Ribaltatore".COut.Ribaltatore.PlusLsSwReached OR "A0301_Ribaltatore".Ax.DataIn.LS_Minus OR "A0301_Ribaltatore".Ax.DataIn.LS_Plus) AND #MB3_Decoder.OpRunning THEN
       "A0301_Ribaltatore".HMI.OP_Sel_Pos1 := FALSE;
       #MB3_Decoder.OpDone := TRUE;
   END_IF;
END_REGION

REGION Network 16: MB3 Code 6010 - Rotazione Ribalta - OP POS2
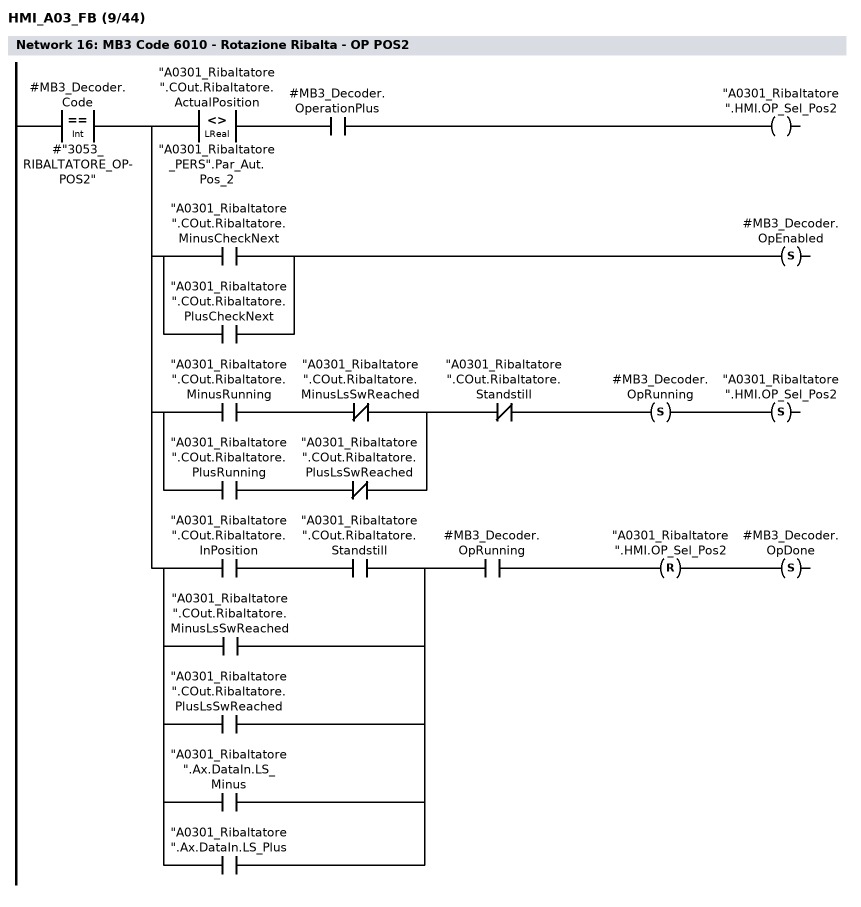
   RUNG wire#powerrail
      { S7_Templates := "SrcType := Int" } EQ_Contact(in1 := #MB3_Decoder.Code, in2 := #"3053_RIBALTATORE_OP-POS2")
      wire#w1
      { S7_Templates := "SrcType := LReal" } NE_Contact(in1 := "A0301_Ribaltatore".COut.Ribaltatore.ActualPosition, in2 := "A0301_Ribaltatore_PERS".Par_Aut.Pos_2)
      Contact( #MB3_Decoder.OperationPlus )
      Coil( "A0301_Ribaltatore".HMI.OP_Sel_Pos2 )
   END_RUNG
   RUNG wire#w1
      Contact( "A0301_Ribaltatore".COut.Ribaltatore.MinusCheckNext )
      wire#w2
      S_Coil( #MB3_Decoder.OpEnabled )
   END_RUNG
   RUNG wire#w1
      Contact( "A0301_Ribaltatore".COut.Ribaltatore.PlusCheckNext )
   END_RUNG wire#w2
   RUNG wire#w1
      Contact( "A0301_Ribaltatore".COut.Ribaltatore.MinusRunning )
      I_Contact( "A0301_Ribaltatore".COut.Ribaltatore.MinusLsSwReached )
      wire#w3
      I_Contact( "A0301_Ribaltatore".COut.Ribaltatore.Standstill )
      S_Coil( #MB3_Decoder.OpRunning )
      S_Coil( "A0301_Ribaltatore".HMI.OP_Sel_Pos2 )
   END_RUNG
   RUNG wire#w1
      Contact( "A0301_Ribaltatore".COut.Ribaltatore.PlusRunning )
      I_Contact( "A0301_Ribaltatore".COut.Ribaltatore.PlusLsSwReached )
   END_RUNG wire#w3
   RUNG wire#w1
      Contact( "A0301_Ribaltatore".COut.Ribaltatore.InPosition )
      Contact( "A0301_Ribaltatore".COut.Ribaltatore.Standstill )
      wire#w4
      Contact( #MB3_Decoder.OpRunning )
      R_Coil( "A0301_Ribaltatore".HMI.OP_Sel_Pos2 )
      S_Coil( #MB3_Decoder.OpDone )
   END_RUNG
   RUNG wire#w1
      Contact( "A0301_Ribaltatore".COut.Ribaltatore.MinusLsSwReached )
   END_RUNG wire#w4
   RUNG wire#w1
      Contact( "A0301_Ribaltatore".COut.Ribaltatore.PlusLsSwReached )
   END_RUNG wire#w4
   RUNG wire#w1
      Contact( "A0301_Ribaltatore".Ax.DataIn.LS_Minus )
   END_RUNG wire#w4
   RUNG wire#w1
      Contact( "A0301_Ribaltatore".Ax.DataIn.LS_Plus )
   END_RUNG wire#w4
   // the same network as SCL:
   #_w1 := #MB3_Decoder.Code = #"3053_RIBALTATORE_OP-POS2";
   "A0301_Ribaltatore".HMI.OP_Sel_Pos2 := #_w1 AND ("A0301_Ribaltatore".COut.Ribaltatore.ActualPosition <> "A0301_Ribaltatore_PERS".Par_Aut.Pos_2) AND #MB3_Decoder.OperationPlus;
   IF #_w1 AND ("A0301_Ribaltatore".COut.Ribaltatore.MinusCheckNext OR "A0301_Ribaltatore".COut.Ribaltatore.PlusCheckNext) THEN
       #MB3_Decoder.OpEnabled := TRUE;
   END_IF;
   IF #_w1 AND (("A0301_Ribaltatore".COut.Ribaltatore.MinusRunning AND NOT "A0301_Ribaltatore".COut.Ribaltatore.MinusLsSwReached) OR ("A0301_Ribaltatore".COut.Ribaltatore.PlusRunning AND NOT "A0301_Ribaltatore".COut.Ribaltatore.PlusLsSwReached)) AND NOT "A0301_Ribaltatore".COut.Ribaltatore.Standstill THEN
       #MB3_Decoder.OpRunning := TRUE;
       "A0301_Ribaltatore".HMI.OP_Sel_Pos2 := TRUE;
   END_IF;
   IF #_w1 AND (("A0301_Ribaltatore".COut.Ribaltatore.InPosition AND "A0301_Ribaltatore".COut.Ribaltatore.Standstill) OR "A0301_Ribaltatore".COut.Ribaltatore.MinusLsSwReached OR "A0301_Ribaltatore".COut.Ribaltatore.PlusLsSwReached OR "A0301_Ribaltatore".Ax.DataIn.LS_Minus OR "A0301_Ribaltatore".Ax.DataIn.LS_Plus) AND #MB3_Decoder.OpRunning THEN
       "A0301_Ribaltatore".HMI.OP_Sel_Pos2 := FALSE;
       #MB3_Decoder.OpDone := TRUE;
   END_IF;
END_REGION

REGION Network 17: MB3 Code 6011 - Rotazione Ribalta - OP POS3
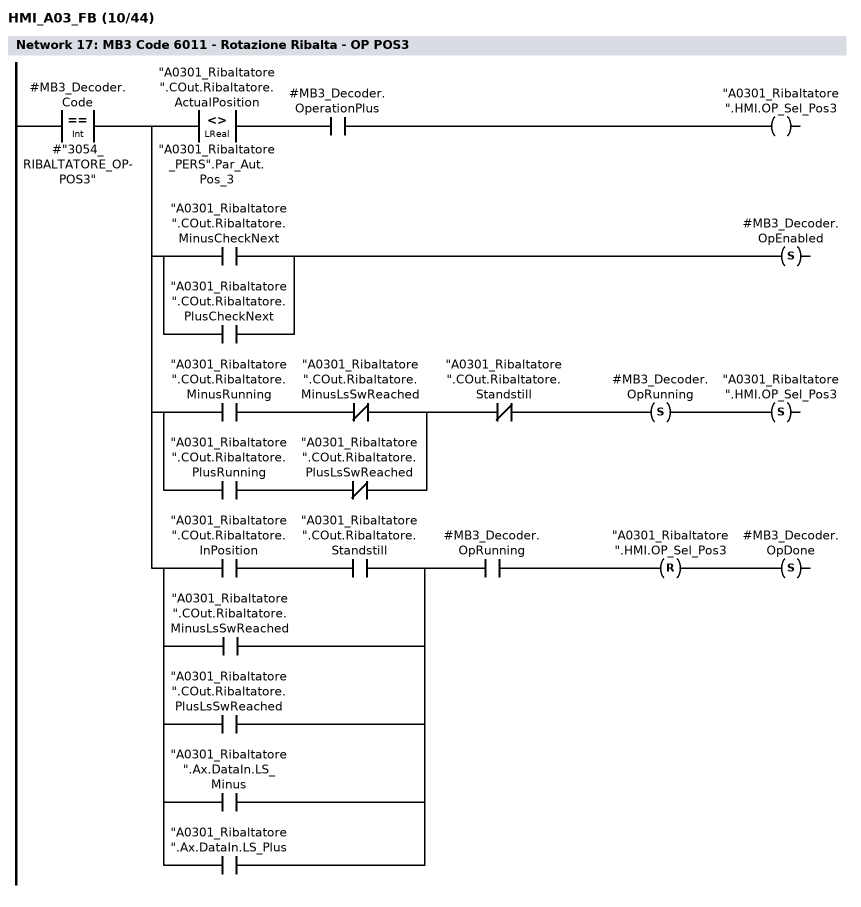
   RUNG wire#powerrail
      { S7_Templates := "SrcType := Int" } EQ_Contact(in1 := #MB3_Decoder.Code, in2 := #"3054_RIBALTATORE_OP-POS3")
      wire#w1
      { S7_Templates := "SrcType := LReal" } NE_Contact(in1 := "A0301_Ribaltatore".COut.Ribaltatore.ActualPosition, in2 := "A0301_Ribaltatore_PERS".Par_Aut.Pos_3)
      Contact( #MB3_Decoder.OperationPlus )
      Coil( "A0301_Ribaltatore".HMI.OP_Sel_Pos3 )
   END_RUNG
   RUNG wire#w1
      Contact( "A0301_Ribaltatore".COut.Ribaltatore.MinusCheckNext )
      wire#w2
      S_Coil( #MB3_Decoder.OpEnabled )
   END_RUNG
   RUNG wire#w1
      Contact( "A0301_Ribaltatore".COut.Ribaltatore.PlusCheckNext )
   END_RUNG wire#w2
   RUNG wire#w1
      Contact( "A0301_Ribaltatore".COut.Ribaltatore.MinusRunning )
      I_Contact( "A0301_Ribaltatore".COut.Ribaltatore.MinusLsSwReached )
      wire#w3
      I_Contact( "A0301_Ribaltatore".COut.Ribaltatore.Standstill )
      S_Coil( #MB3_Decoder.OpRunning )
      S_Coil( "A0301_Ribaltatore".HMI.OP_Sel_Pos3 )
   END_RUNG
   RUNG wire#w1
      Contact( "A0301_Ribaltatore".COut.Ribaltatore.PlusRunning )
      I_Contact( "A0301_Ribaltatore".COut.Ribaltatore.PlusLsSwReached )
   END_RUNG wire#w3
   RUNG wire#w1
      Contact( "A0301_Ribaltatore".COut.Ribaltatore.InPosition )
      Contact( "A0301_Ribaltatore".COut.Ribaltatore.Standstill )
      wire#w4
      Contact( #MB3_Decoder.OpRunning )
      R_Coil( "A0301_Ribaltatore".HMI.OP_Sel_Pos3 )
      S_Coil( #MB3_Decoder.OpDone )
   END_RUNG
   RUNG wire#w1
      Contact( "A0301_Ribaltatore".COut.Ribaltatore.MinusLsSwReached )
   END_RUNG wire#w4
   RUNG wire#w1
      Contact( "A0301_Ribaltatore".COut.Ribaltatore.PlusLsSwReached )
   END_RUNG wire#w4
   RUNG wire#w1
      Contact( "A0301_Ribaltatore".Ax.DataIn.LS_Minus )
   END_RUNG wire#w4
   RUNG wire#w1
      Contact( "A0301_Ribaltatore".Ax.DataIn.LS_Plus )
   END_RUNG wire#w4
   // the same network as SCL:
   #_w1 := #MB3_Decoder.Code = #"3054_RIBALTATORE_OP-POS3";
   "A0301_Ribaltatore".HMI.OP_Sel_Pos3 := #_w1 AND ("A0301_Ribaltatore".COut.Ribaltatore.ActualPosition <> "A0301_Ribaltatore_PERS".Par_Aut.Pos_3) AND #MB3_Decoder.OperationPlus;
   IF #_w1 AND ("A0301_Ribaltatore".COut.Ribaltatore.MinusCheckNext OR "A0301_Ribaltatore".COut.Ribaltatore.PlusCheckNext) THEN
       #MB3_Decoder.OpEnabled := TRUE;
   END_IF;
   IF #_w1 AND (("A0301_Ribaltatore".COut.Ribaltatore.MinusRunning AND NOT "A0301_Ribaltatore".COut.Ribaltatore.MinusLsSwReached) OR ("A0301_Ribaltatore".COut.Ribaltatore.PlusRunning AND NOT "A0301_Ribaltatore".COut.Ribaltatore.PlusLsSwReached)) AND NOT "A0301_Ribaltatore".COut.Ribaltatore.Standstill THEN
       #MB3_Decoder.OpRunning := TRUE;
       "A0301_Ribaltatore".HMI.OP_Sel_Pos3 := TRUE;
   END_IF;
   IF #_w1 AND (("A0301_Ribaltatore".COut.Ribaltatore.InPosition AND "A0301_Ribaltatore".COut.Ribaltatore.Standstill) OR "A0301_Ribaltatore".COut.Ribaltatore.MinusLsSwReached OR "A0301_Ribaltatore".COut.Ribaltatore.PlusLsSwReached OR "A0301_Ribaltatore".Ax.DataIn.LS_Minus OR "A0301_Ribaltatore".Ax.DataIn.LS_Plus) AND #MB3_Decoder.OpRunning THEN
       "A0301_Ribaltatore".HMI.OP_Sel_Pos3 := FALSE;
       #MB3_Decoder.OpDone := TRUE;
   END_IF;
END_REGION

REGION Network 18: MB3 Code 3041 - Fermi P4
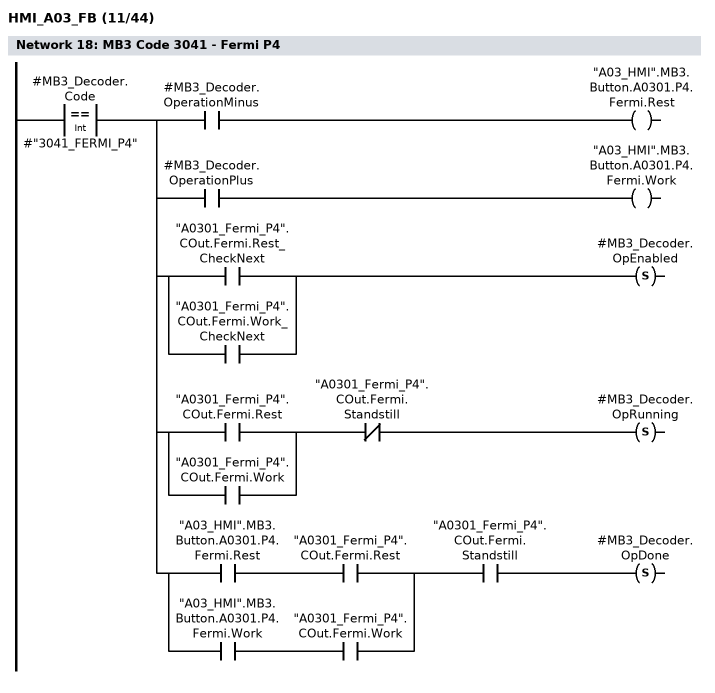
   RUNG wire#powerrail
      { S7_Templates := "SrcType := Int" } EQ_Contact(in1 := #MB3_Decoder.Code, in2 := #"3041_FERMI_P4")
      wire#w1
      Contact( #MB3_Decoder.OperationMinus )
      Coil( "A03_HMI".MB3.Button.A0301.P4.Fermi.Rest )
   END_RUNG
   RUNG wire#w1
      Contact( #MB3_Decoder.OperationPlus )
      Coil( "A03_HMI".MB3.Button.A0301.P4.Fermi.Work )
   END_RUNG
   RUNG wire#w1
      Contact( "A0301_Fermi_P4".COut.Fermi.Rest_CheckNext )
      wire#w2
      S_Coil( #MB3_Decoder.OpEnabled )
   END_RUNG
   RUNG wire#w1
      Contact( "A0301_Fermi_P4".COut.Fermi.Work_CheckNext )
   END_RUNG wire#w2
   RUNG wire#w1
      Contact( "A0301_Fermi_P4".COut.Fermi.Rest )
      wire#w3
      I_Contact( "A0301_Fermi_P4".COut.Fermi.Standstill )
      S_Coil( #MB3_Decoder.OpRunning )
   END_RUNG
   RUNG wire#w1
      Contact( "A0301_Fermi_P4".COut.Fermi.Work )
   END_RUNG wire#w3
   RUNG wire#w1
      Contact( "A03_HMI".MB3.Button.A0301.P4.Fermi.Rest )
      Contact( "A0301_Fermi_P4".COut.Fermi.Rest )
      wire#w4
      Contact( "A0301_Fermi_P4".COut.Fermi.Standstill )
      S_Coil( #MB3_Decoder.OpDone )
   END_RUNG
   RUNG wire#w1
      Contact( "A03_HMI".MB3.Button.A0301.P4.Fermi.Work )
      Contact( "A0301_Fermi_P4".COut.Fermi.Work )
   END_RUNG wire#w4
   // the same network as SCL:
   #_w1 := #MB3_Decoder.Code = #"3041_FERMI_P4";
   "A03_HMI".MB3.Button.A0301.P4.Fermi.Rest := #_w1 AND #MB3_Decoder.OperationMinus;
   "A03_HMI".MB3.Button.A0301.P4.Fermi.Work := #_w1 AND #MB3_Decoder.OperationPlus;
   IF #_w1 AND ("A0301_Fermi_P4".COut.Fermi.Rest_CheckNext OR "A0301_Fermi_P4".COut.Fermi.Work_CheckNext) THEN
       #MB3_Decoder.OpEnabled := TRUE;
   END_IF;
   IF #_w1 AND ("A0301_Fermi_P4".COut.Fermi.Rest OR "A0301_Fermi_P4".COut.Fermi.Work) AND NOT "A0301_Fermi_P4".COut.Fermi.Standstill THEN
       #MB3_Decoder.OpRunning := TRUE;
   END_IF;
   IF #_w1 AND (("A03_HMI".MB3.Button.A0301.P4.Fermi.Rest AND "A0301_Fermi_P4".COut.Fermi.Rest) OR ("A03_HMI".MB3.Button.A0301.P4.Fermi.Work AND "A0301_Fermi_P4".COut.Fermi.Work)) AND "A0301_Fermi_P4".COut.Fermi.Standstill THEN
       #MB3_Decoder.OpDone := TRUE;
   END_IF;
END_REGION

REGION Network 19: MB3 Code 3042 - P5 - Spintore Laterale-Vrt
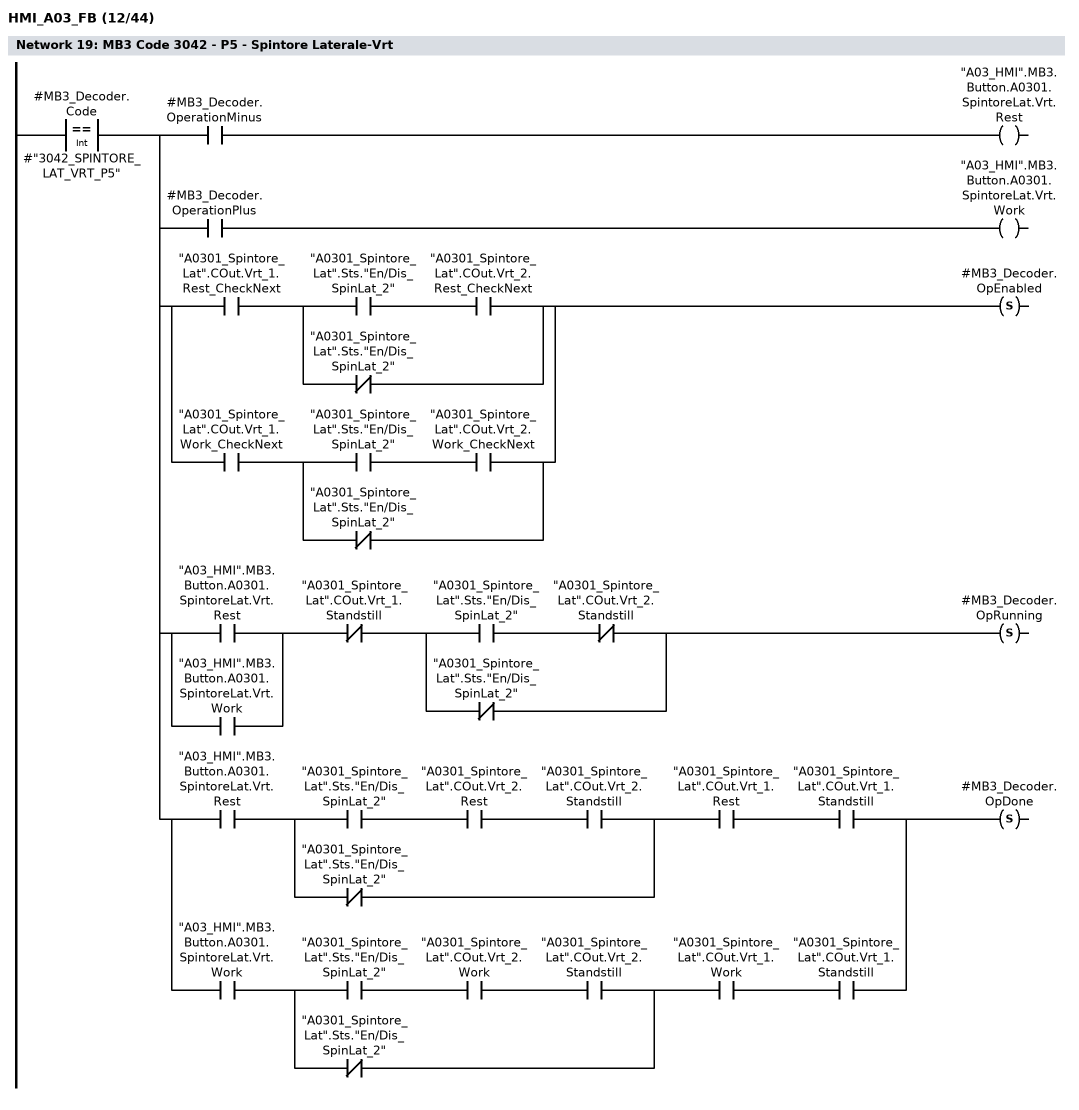
   RUNG wire#powerrail
      { S7_Templates := "SrcType := Int" } EQ_Contact(in1 := #MB3_Decoder.Code, in2 := #"3042_SPINTORE_LAT_VRT_P5")
      wire#w1
      Contact( #MB3_Decoder.OperationMinus )
      Coil( "A03_HMI".MB3.Button.A0301.SpintoreLat.Vrt.Rest )
   END_RUNG
   RUNG wire#w1
      Contact( #MB3_Decoder.OperationPlus )
      Coil( "A03_HMI".MB3.Button.A0301.SpintoreLat.Vrt.Work )
   END_RUNG
   RUNG wire#w1
      Contact( "A0301_Spintore_Lat".COut.Vrt_1.Rest_CheckNext )
      wire#w2
      Contact( "A0301_Spintore_Lat".Sts."En/Dis_SpinLat_2" )
      Contact( "A0301_Spintore_Lat".COut.Vrt_2.Rest_CheckNext )
      wire#w3
      S_Coil( #MB3_Decoder.OpEnabled )
   END_RUNG
   RUNG wire#w2
      I_Contact( "A0301_Spintore_Lat".Sts."En/Dis_SpinLat_2" )
   END_RUNG wire#w3
   RUNG wire#w1
      Contact( "A0301_Spintore_Lat".COut.Vrt_1.Work_CheckNext )
      wire#w4
      Contact( "A0301_Spintore_Lat".Sts."En/Dis_SpinLat_2" )
      Contact( "A0301_Spintore_Lat".COut.Vrt_2.Work_CheckNext )
   END_RUNG wire#w3
   RUNG wire#w4
      I_Contact( "A0301_Spintore_Lat".Sts."En/Dis_SpinLat_2" )
   END_RUNG wire#w3
   RUNG wire#w1
      Contact( "A03_HMI".MB3.Button.A0301.SpintoreLat.Vrt.Rest )
      wire#w5
      I_Contact( "A0301_Spintore_Lat".COut.Vrt_1.Standstill )
      wire#w6
      Contact( "A0301_Spintore_Lat".Sts."En/Dis_SpinLat_2" )
      I_Contact( "A0301_Spintore_Lat".COut.Vrt_2.Standstill )
      wire#w7
      S_Coil( #MB3_Decoder.OpRunning )
   END_RUNG
   RUNG wire#w1
      Contact( "A03_HMI".MB3.Button.A0301.SpintoreLat.Vrt.Work )
   END_RUNG wire#w5
   RUNG wire#w6
      I_Contact( "A0301_Spintore_Lat".Sts."En/Dis_SpinLat_2" )
   END_RUNG wire#w7
   RUNG wire#w1
      Contact( "A03_HMI".MB3.Button.A0301.SpintoreLat.Vrt.Rest )
      wire#w8
      Contact( "A0301_Spintore_Lat".Sts."En/Dis_SpinLat_2" )
      Contact( "A0301_Spintore_Lat".COut.Vrt_2.Rest )
      Contact( "A0301_Spintore_Lat".COut.Vrt_2.Standstill )
      wire#w9
      Contact( "A0301_Spintore_Lat".COut.Vrt_1.Rest )
      Contact( "A0301_Spintore_Lat".COut.Vrt_1.Standstill )
      wire#w10
      S_Coil( #MB3_Decoder.OpDone )
   END_RUNG
   RUNG wire#w8
      I_Contact( "A0301_Spintore_Lat".Sts."En/Dis_SpinLat_2" )
   END_RUNG wire#w9
   RUNG wire#w1
      Contact( "A03_HMI".MB3.Button.A0301.SpintoreLat.Vrt.Work )
      wire#w11
      Contact( "A0301_Spintore_Lat".Sts."En/Dis_SpinLat_2" )
      Contact( "A0301_Spintore_Lat".COut.Vrt_2.Work )
      Contact( "A0301_Spintore_Lat".COut.Vrt_2.Standstill )
      wire#w12
      Contact( "A0301_Spintore_Lat".COut.Vrt_1.Work )
      Contact( "A0301_Spintore_Lat".COut.Vrt_1.Standstill )
   END_RUNG wire#w10
   RUNG wire#w11
      I_Contact( "A0301_Spintore_Lat".Sts."En/Dis_SpinLat_2" )
   END_RUNG wire#w12
   // the same network as SCL:
   #_w1 := #MB3_Decoder.Code = #"3042_SPINTORE_LAT_VRT_P5";
   "A03_HMI".MB3.Button.A0301.SpintoreLat.Vrt.Rest := #_w1 AND #MB3_Decoder.OperationMinus;
   "A03_HMI".MB3.Button.A0301.SpintoreLat.Vrt.Work := #_w1 AND #MB3_Decoder.OperationPlus;
   IF #_w1 AND (("A0301_Spintore_Lat".COut.Vrt_1.Rest_CheckNext AND (("A0301_Spintore_Lat".Sts."En/Dis_SpinLat_2" AND "A0301_Spintore_Lat".COut.Vrt_2.Rest_CheckNext) OR NOT "A0301_Spintore_Lat".Sts."En/Dis_SpinLat_2")) OR ("A0301_Spintore_Lat".COut.Vrt_1.Work_CheckNext AND (("A0301_Spintore_Lat".Sts."En/Dis_SpinLat_2" AND "A0301_Spintore_Lat".COut.Vrt_2.Work_CheckNext) OR NOT "A0301_Spintore_Lat".Sts."En/Dis_SpinLat_2"))) THEN
       #MB3_Decoder.OpEnabled := TRUE;
   END_IF;
   IF #_w1 AND ("A03_HMI".MB3.Button.A0301.SpintoreLat.Vrt.Rest OR "A03_HMI".MB3.Button.A0301.SpintoreLat.Vrt.Work) AND NOT "A0301_Spintore_Lat".COut.Vrt_1.Standstill AND (("A0301_Spintore_Lat".Sts."En/Dis_SpinLat_2" AND NOT "A0301_Spintore_Lat".COut.Vrt_2.Standstill) OR NOT "A0301_Spintore_Lat".Sts."En/Dis_SpinLat_2") THEN
       #MB3_Decoder.OpRunning := TRUE;
   END_IF;
   IF #_w1 AND (("A03_HMI".MB3.Button.A0301.SpintoreLat.Vrt.Rest AND (("A0301_Spintore_Lat".Sts."En/Dis_SpinLat_2" AND "A0301_Spintore_Lat".COut.Vrt_2.Rest AND "A0301_Spintore_Lat".COut.Vrt_2.Standstill) OR NOT "A0301_Spintore_Lat".Sts."En/Dis_SpinLat_2") AND "A0301_Spintore_Lat".COut.Vrt_1.Rest AND "A0301_Spintore_Lat".COut.Vrt_1.Standstill) OR ("A03_HMI".MB3.Button.A0301.SpintoreLat.Vrt.Work AND (("A0301_Spintore_Lat".Sts."En/Dis_SpinLat_2" AND "A0301_Spintore_Lat".COut.Vrt_2.Work AND "A0301_Spintore_Lat".COut.Vrt_2.Standstill) OR NOT "A0301_Spintore_Lat".Sts."En/Dis_SpinLat_2") AND "A0301_Spintore_Lat".COut.Vrt_1.Work AND "A0301_Spintore_Lat".COut.Vrt_1.Standstill)) THEN
       #MB3_Decoder.OpDone := TRUE;
   END_IF;
END_REGION

REGION Network 20: MB3 Code 3043 - P5 - Spintore Laterale-Orz
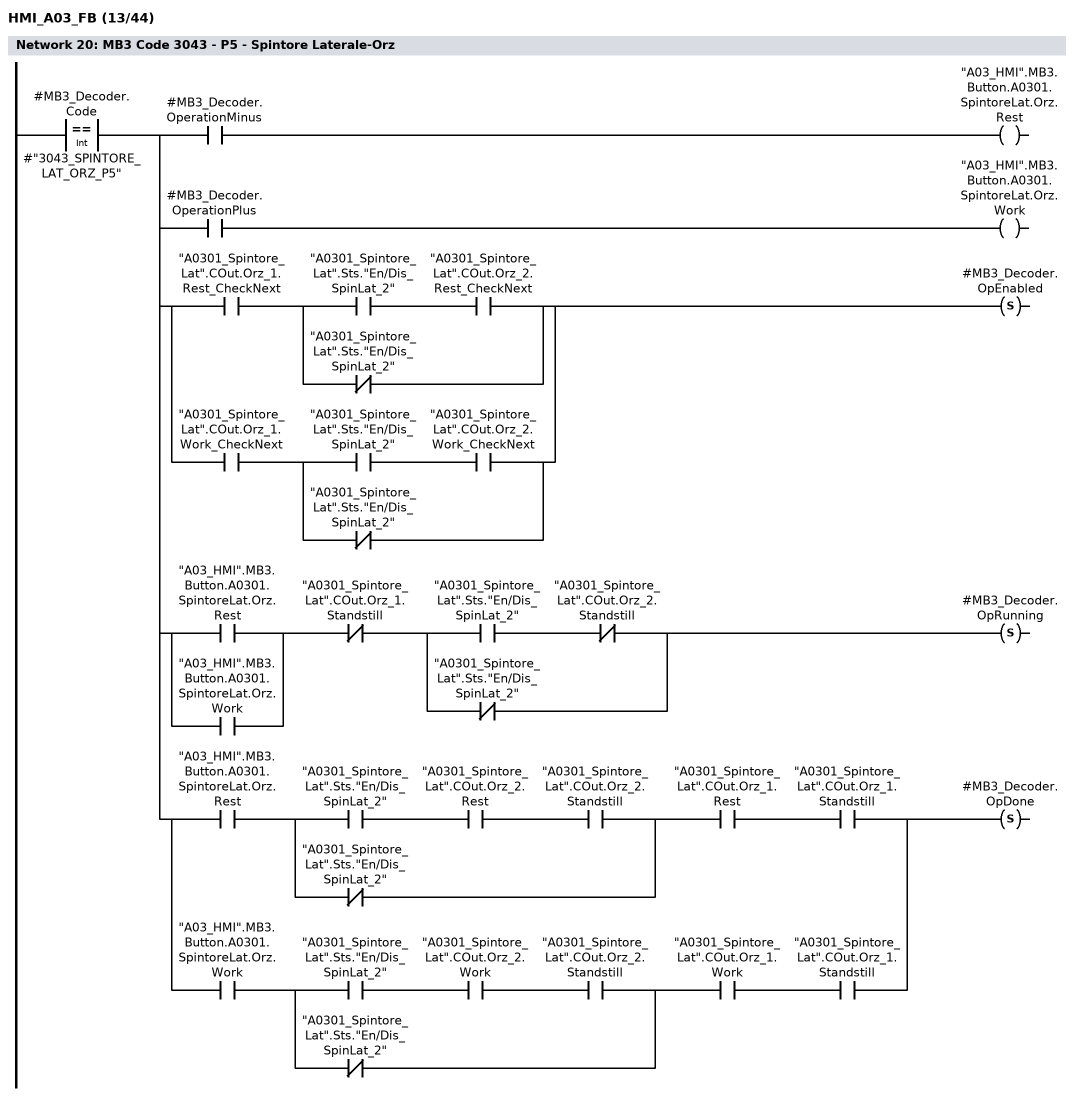
   RUNG wire#powerrail
      { S7_Templates := "SrcType := Int" } EQ_Contact(in1 := #MB3_Decoder.Code, in2 := #"3043_SPINTORE_LAT_ORZ_P5")
      wire#w1
      Contact( #MB3_Decoder.OperationMinus )
      Coil( "A03_HMI".MB3.Button.A0301.SpintoreLat.Orz.Rest )
   END_RUNG
   RUNG wire#w1
      Contact( #MB3_Decoder.OperationPlus )
      Coil( "A03_HMI".MB3.Button.A0301.SpintoreLat.Orz.Work )
   END_RUNG
   RUNG wire#w1
      Contact( "A0301_Spintore_Lat".COut.Orz_1.Rest_CheckNext )
      wire#w2
      Contact( "A0301_Spintore_Lat".Sts."En/Dis_SpinLat_2" )
      Contact( "A0301_Spintore_Lat".COut.Orz_2.Rest_CheckNext )
      wire#w3
      S_Coil( #MB3_Decoder.OpEnabled )
   END_RUNG
   RUNG wire#w2
      I_Contact( "A0301_Spintore_Lat".Sts."En/Dis_SpinLat_2" )
   END_RUNG wire#w3
   RUNG wire#w1
      Contact( "A0301_Spintore_Lat".COut.Orz_1.Work_CheckNext )
      wire#w4
      Contact( "A0301_Spintore_Lat".Sts."En/Dis_SpinLat_2" )
      Contact( "A0301_Spintore_Lat".COut.Orz_2.Work_CheckNext )
   END_RUNG wire#w3
   RUNG wire#w4
      I_Contact( "A0301_Spintore_Lat".Sts."En/Dis_SpinLat_2" )
   END_RUNG wire#w3
   RUNG wire#w1
      Contact( "A03_HMI".MB3.Button.A0301.SpintoreLat.Orz.Rest )
      wire#w5
      I_Contact( "A0301_Spintore_Lat".COut.Orz_1.Standstill )
      wire#w6
      Contact( "A0301_Spintore_Lat".Sts."En/Dis_SpinLat_2" )
      I_Contact( "A0301_Spintore_Lat".COut.Orz_2.Standstill )
      wire#w7
      S_Coil( #MB3_Decoder.OpRunning )
   END_RUNG
   RUNG wire#w1
      Contact( "A03_HMI".MB3.Button.A0301.SpintoreLat.Orz.Work )
   END_RUNG wire#w5
   RUNG wire#w6
      I_Contact( "A0301_Spintore_Lat".Sts."En/Dis_SpinLat_2" )
   END_RUNG wire#w7
   RUNG wire#w1
      Contact( "A03_HMI".MB3.Button.A0301.SpintoreLat.Orz.Rest )
      wire#w8
      Contact( "A0301_Spintore_Lat".Sts."En/Dis_SpinLat_2" )
      Contact( "A0301_Spintore_Lat".COut.Orz_2.Rest )
      Contact( "A0301_Spintore_Lat".COut.Orz_2.Standstill )
      wire#w9
      Contact( "A0301_Spintore_Lat".COut.Orz_1.Rest )
      Contact( "A0301_Spintore_Lat".COut.Orz_1.Standstill )
      wire#w10
      S_Coil( #MB3_Decoder.OpDone )
   END_RUNG
   RUNG wire#w8
      I_Contact( "A0301_Spintore_Lat".Sts."En/Dis_SpinLat_2" )
   END_RUNG wire#w9
   RUNG wire#w1
      Contact( "A03_HMI".MB3.Button.A0301.SpintoreLat.Orz.Work )
      wire#w11
      Contact( "A0301_Spintore_Lat".Sts."En/Dis_SpinLat_2" )
      Contact( "A0301_Spintore_Lat".COut.Orz_2.Work )
      Contact( "A0301_Spintore_Lat".COut.Orz_2.Standstill )
      wire#w12
      Contact( "A0301_Spintore_Lat".COut.Orz_1.Work )
      Contact( "A0301_Spintore_Lat".COut.Orz_1.Standstill )
   END_RUNG wire#w10
   RUNG wire#w11
      I_Contact( "A0301_Spintore_Lat".Sts."En/Dis_SpinLat_2" )
   END_RUNG wire#w12
   // the same network as SCL:
   #_w1 := #MB3_Decoder.Code = #"3043_SPINTORE_LAT_ORZ_P5";
   "A03_HMI".MB3.Button.A0301.SpintoreLat.Orz.Rest := #_w1 AND #MB3_Decoder.OperationMinus;
   "A03_HMI".MB3.Button.A0301.SpintoreLat.Orz.Work := #_w1 AND #MB3_Decoder.OperationPlus;
   IF #_w1 AND (("A0301_Spintore_Lat".COut.Orz_1.Rest_CheckNext AND (("A0301_Spintore_Lat".Sts."En/Dis_SpinLat_2" AND "A0301_Spintore_Lat".COut.Orz_2.Rest_CheckNext) OR NOT "A0301_Spintore_Lat".Sts."En/Dis_SpinLat_2")) OR ("A0301_Spintore_Lat".COut.Orz_1.Work_CheckNext AND (("A0301_Spintore_Lat".Sts."En/Dis_SpinLat_2" AND "A0301_Spintore_Lat".COut.Orz_2.Work_CheckNext) OR NOT "A0301_Spintore_Lat".Sts."En/Dis_SpinLat_2"))) THEN
       #MB3_Decoder.OpEnabled := TRUE;
   END_IF;
   IF #_w1 AND ("A03_HMI".MB3.Button.A0301.SpintoreLat.Orz.Rest OR "A03_HMI".MB3.Button.A0301.SpintoreLat.Orz.Work) AND NOT "A0301_Spintore_Lat".COut.Orz_1.Standstill AND (("A0301_Spintore_Lat".Sts."En/Dis_SpinLat_2" AND NOT "A0301_Spintore_Lat".COut.Orz_2.Standstill) OR NOT "A0301_Spintore_Lat".Sts."En/Dis_SpinLat_2") THEN
       #MB3_Decoder.OpRunning := TRUE;
   END_IF;
   IF #_w1 AND (("A03_HMI".MB3.Button.A0301.SpintoreLat.Orz.Rest AND (("A0301_Spintore_Lat".Sts."En/Dis_SpinLat_2" AND "A0301_Spintore_Lat".COut.Orz_2.Rest AND "A0301_Spintore_Lat".COut.Orz_2.Standstill) OR NOT "A0301_Spintore_Lat".Sts."En/Dis_SpinLat_2") AND "A0301_Spintore_Lat".COut.Orz_1.Rest AND "A0301_Spintore_Lat".COut.Orz_1.Standstill) OR ("A03_HMI".MB3.Button.A0301.SpintoreLat.Orz.Work AND (("A0301_Spintore_Lat".Sts."En/Dis_SpinLat_2" AND "A0301_Spintore_Lat".COut.Orz_2.Work AND "A0301_Spintore_Lat".COut.Orz_2.Standstill) OR NOT "A0301_Spintore_Lat".Sts."En/Dis_SpinLat_2") AND "A0301_Spintore_Lat".COut.Orz_1.Work AND "A0301_Spintore_Lat".COut.Orz_1.Standstill)) THEN
       #MB3_Decoder.OpDone := TRUE;
   END_IF;
END_REGION

REGION Network 21: MB3 Code 3045 - P5 - Spintore Laterale-OP
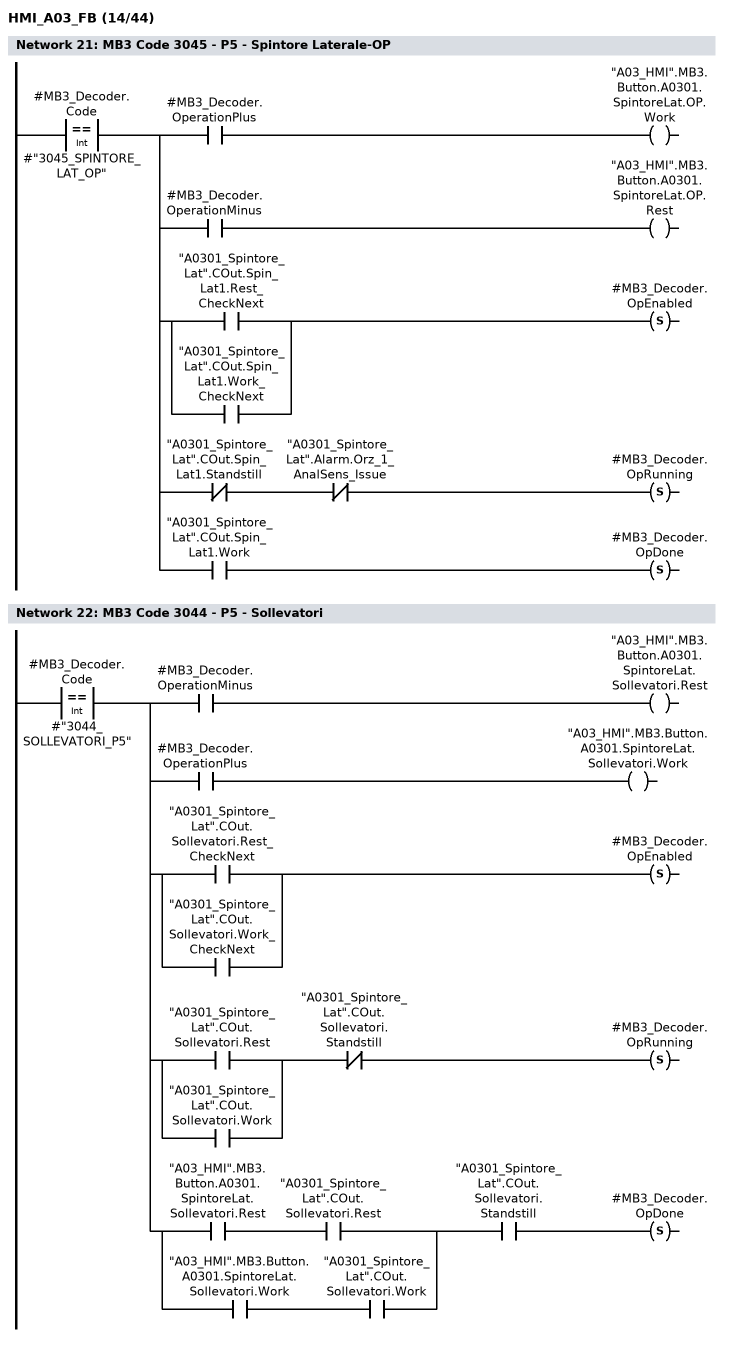
   RUNG wire#powerrail
      { S7_Templates := "SrcType := Int" } EQ_Contact(in1 := #MB3_Decoder.Code, in2 := #"3045_SPINTORE_LAT_OP")
      wire#w1
      Contact( #MB3_Decoder.OperationPlus )
      Coil( "A03_HMI".MB3.Button.A0301.SpintoreLat.OP.Work )
   END_RUNG
   RUNG wire#w1
      Contact( #MB3_Decoder.OperationMinus )
      Coil( "A03_HMI".MB3.Button.A0301.SpintoreLat.OP.Rest )
   END_RUNG
   RUNG wire#w1
      Contact( "A0301_Spintore_Lat".COut.Spin_Lat1.Rest_CheckNext )
      wire#w2
      S_Coil( #MB3_Decoder.OpEnabled )
   END_RUNG
   RUNG wire#w1
      Contact( "A0301_Spintore_Lat".COut.Spin_Lat1.Work_CheckNext )
   END_RUNG wire#w2
   RUNG wire#w1
      I_Contact( "A0301_Spintore_Lat".COut.Spin_Lat1.Standstill )
      I_Contact( "A0301_Spintore_Lat".Alarm.Orz_1_AnalSens_Issue )
      S_Coil( #MB3_Decoder.OpRunning )
   END_RUNG
   RUNG wire#w1
      Contact( "A0301_Spintore_Lat".COut.Spin_Lat1.Work )
      S_Coil( #MB3_Decoder.OpDone )
   END_RUNG
   // the same network as SCL:
   #_w1 := #MB3_Decoder.Code = #"3045_SPINTORE_LAT_OP";
   "A03_HMI".MB3.Button.A0301.SpintoreLat.OP.Work := #_w1 AND #MB3_Decoder.OperationPlus;
   "A03_HMI".MB3.Button.A0301.SpintoreLat.OP.Rest := #_w1 AND #MB3_Decoder.OperationMinus;
   IF #_w1 AND ("A0301_Spintore_Lat".COut.Spin_Lat1.Rest_CheckNext OR "A0301_Spintore_Lat".COut.Spin_Lat1.Work_CheckNext) THEN
       #MB3_Decoder.OpEnabled := TRUE;
   END_IF;
   IF #_w1 AND NOT "A0301_Spintore_Lat".COut.Spin_Lat1.Standstill AND NOT "A0301_Spintore_Lat".Alarm.Orz_1_AnalSens_Issue THEN
       #MB3_Decoder.OpRunning := TRUE;
   END_IF;
   IF #_w1 AND "A0301_Spintore_Lat".COut.Spin_Lat1.Work THEN #MB3_Decoder.OpDone := TRUE; END_IF;
END_REGION

REGION Network 22: MB3 Code 3044 - P5 - Sollevatori
   RUNG wire#powerrail
      { S7_Templates := "SrcType := Int" } EQ_Contact(in1 := #MB3_Decoder.Code, in2 := #"3044_SOLLEVATORI_P5")
      wire#w1
      Contact( #MB3_Decoder.OperationMinus )
      Coil( "A03_HMI".MB3.Button.A0301.SpintoreLat.Sollevatori.Rest )
   END_RUNG
   RUNG wire#w1
      Contact( #MB3_Decoder.OperationPlus )
      Coil( "A03_HMI".MB3.Button.A0301.SpintoreLat.Sollevatori.Work )
   END_RUNG
   RUNG wire#w1
      Contact( "A0301_Spintore_Lat".COut.Sollevatori.Rest_CheckNext )
      wire#w2
      S_Coil( #MB3_Decoder.OpEnabled )
   END_RUNG
   RUNG wire#w1
      Contact( "A0301_Spintore_Lat".COut.Sollevatori.Work_CheckNext )
   END_RUNG wire#w2
   RUNG wire#w1
      Contact( "A0301_Spintore_Lat".COut.Sollevatori.Rest )
      wire#w3
      I_Contact( "A0301_Spintore_Lat".COut.Sollevatori.Standstill )
      S_Coil( #MB3_Decoder.OpRunning )
   END_RUNG
   RUNG wire#w1
      Contact( "A0301_Spintore_Lat".COut.Sollevatori.Work )
   END_RUNG wire#w3
   RUNG wire#w1
      Contact( "A03_HMI".MB3.Button.A0301.SpintoreLat.Sollevatori.Rest )
      Contact( "A0301_Spintore_Lat".COut.Sollevatori.Rest )
      wire#w4
      Contact( "A0301_Spintore_Lat".COut.Sollevatori.Standstill )
      S_Coil( #MB3_Decoder.OpDone )
   END_RUNG
   RUNG wire#w1
      Contact( "A03_HMI".MB3.Button.A0301.SpintoreLat.Sollevatori.Work )
      Contact( "A0301_Spintore_Lat".COut.Sollevatori.Work )
   END_RUNG wire#w4
   // the same network as SCL:
   #_w1 := #MB3_Decoder.Code = #"3044_SOLLEVATORI_P5";
   "A03_HMI".MB3.Button.A0301.SpintoreLat.Sollevatori.Rest := #_w1 AND #MB3_Decoder.OperationMinus;
   "A03_HMI".MB3.Button.A0301.SpintoreLat.Sollevatori.Work := #_w1 AND #MB3_Decoder.OperationPlus;
   IF #_w1 AND ("A0301_Spintore_Lat".COut.Sollevatori.Rest_CheckNext OR "A0301_Spintore_Lat".COut.Sollevatori.Work_CheckNext) THEN
       #MB3_Decoder.OpEnabled := TRUE;
   END_IF;
   IF #_w1 AND ("A0301_Spintore_Lat".COut.Sollevatori.Rest OR "A0301_Spintore_Lat".COut.Sollevatori.Work) AND NOT "A0301_Spintore_Lat".COut.Sollevatori.Standstill THEN
       #MB3_Decoder.OpRunning := TRUE;
   END_IF;
   IF #_w1 AND (("A03_HMI".MB3.Button.A0301.SpintoreLat.Sollevatori.Rest AND "A0301_Spintore_Lat".COut.Sollevatori.Rest) OR ("A03_HMI".MB3.Button.A0301.SpintoreLat.Sollevatori.Work AND "A0301_Spintore_Lat".COut.Sollevatori.Work)) AND "A0301_Spintore_Lat".COut.Sollevatori.Standstill THEN
       #MB3_Decoder.OpDone := TRUE;
   END_IF;
END_REGION

REGION Network 23: <<<<<<<<< A0302 STAZIONE 2 >>>>>>>>>>>>>
END_REGION

REGION Network 24: MB3 Code 4001 - Area 03 HU Cytropack
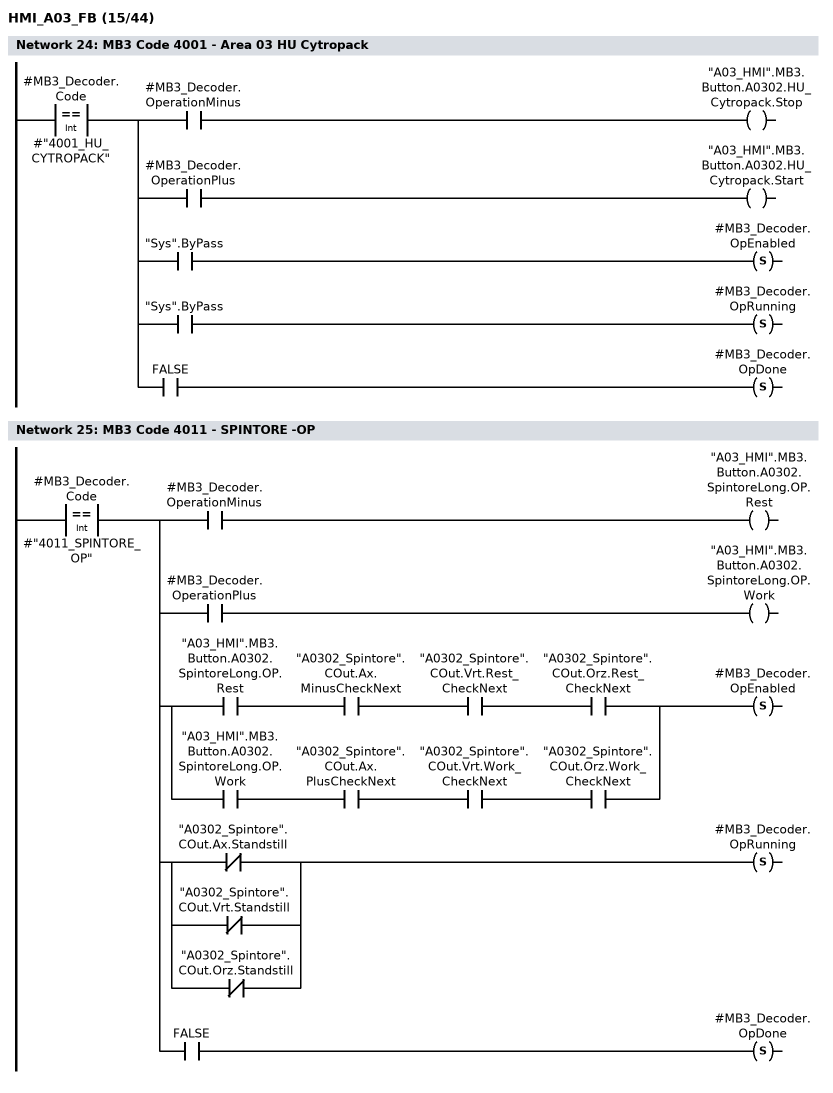
   RUNG wire#powerrail
      { S7_Templates := "SrcType := Int" } EQ_Contact(in1 := #MB3_Decoder.Code, in2 := #"4001_HU_CYTROPACK")
      wire#w1
      Contact( #MB3_Decoder.OperationMinus )
      Coil( "A03_HMI".MB3.Button.A0302.HU_Cytropack.Stop )
   END_RUNG
   RUNG wire#w1
      Contact( #MB3_Decoder.OperationPlus )
      Coil( "A03_HMI".MB3.Button.A0302.HU_Cytropack.Start )
   END_RUNG
   RUNG wire#w1
      Contact( "Sys".ByPass )
      S_Coil( #MB3_Decoder.OpEnabled )
   END_RUNG
   RUNG wire#w1
      Contact( "Sys".ByPass )
      S_Coil( #MB3_Decoder.OpRunning )
   END_RUNG
   RUNG wire#w1
      Contact( FALSE )
      S_Coil( #MB3_Decoder.OpDone )
   END_RUNG
   // the same network as SCL:
   #_w1 := #MB3_Decoder.Code = #"4001_HU_CYTROPACK";
   "A03_HMI".MB3.Button.A0302.HU_Cytropack.Stop := #_w1 AND #MB3_Decoder.OperationMinus;
   "A03_HMI".MB3.Button.A0302.HU_Cytropack.Start := #_w1 AND #MB3_Decoder.OperationPlus;
   IF #_w1 AND "Sys".ByPass THEN
       #MB3_Decoder.OpEnabled := TRUE;
       #MB3_Decoder.OpRunning := TRUE;
   END_IF;
   IF #_w1 AND FALSE THEN #MB3_Decoder.OpDone := TRUE; END_IF;
END_REGION

REGION Network 25: MB3 Code 4011 - SPINTORE -OP
   RUNG wire#powerrail
      { S7_Templates := "SrcType := Int" } EQ_Contact(in1 := #MB3_Decoder.Code, in2 := #"4011_SPINTORE_OP")
      wire#w1
      Contact( #MB3_Decoder.OperationMinus )
      Coil( "A03_HMI".MB3.Button.A0302.SpintoreLong.OP.Rest )
   END_RUNG
   RUNG wire#w1
      Contact( #MB3_Decoder.OperationPlus )
      Coil( "A03_HMI".MB3.Button.A0302.SpintoreLong.OP.Work )
   END_RUNG
   RUNG wire#w1
      Contact( "A03_HMI".MB3.Button.A0302.SpintoreLong.OP.Rest )
      Contact( "A0302_Spintore".COut.Ax.MinusCheckNext )
      Contact( "A0302_Spintore".COut.Vrt.Rest_CheckNext )
      Contact( "A0302_Spintore".COut.Orz.Rest_CheckNext )
      wire#w2
      S_Coil( #MB3_Decoder.OpEnabled )
   END_RUNG
   RUNG wire#w1
      Contact( "A03_HMI".MB3.Button.A0302.SpintoreLong.OP.Work )
      Contact( "A0302_Spintore".COut.Ax.PlusCheckNext )
      Contact( "A0302_Spintore".COut.Vrt.Work_CheckNext )
      Contact( "A0302_Spintore".COut.Orz.Work_CheckNext )
   END_RUNG wire#w2
   RUNG wire#w1
      I_Contact( "A0302_Spintore".COut.Ax.Standstill )
      wire#w3
      S_Coil( #MB3_Decoder.OpRunning )
   END_RUNG
   RUNG wire#w1
      I_Contact( "A0302_Spintore".COut.Vrt.Standstill )
   END_RUNG wire#w3
   RUNG wire#w1
      I_Contact( "A0302_Spintore".COut.Orz.Standstill )
   END_RUNG wire#w3
   RUNG wire#w1
      Contact( FALSE )
      S_Coil( #MB3_Decoder.OpDone )
   END_RUNG
   // the same network as SCL:
   #_w1 := #MB3_Decoder.Code = #"4011_SPINTORE_OP";
   "A03_HMI".MB3.Button.A0302.SpintoreLong.OP.Rest := #_w1 AND #MB3_Decoder.OperationMinus;
   "A03_HMI".MB3.Button.A0302.SpintoreLong.OP.Work := #_w1 AND #MB3_Decoder.OperationPlus;
   IF #_w1 AND (("A03_HMI".MB3.Button.A0302.SpintoreLong.OP.Rest AND "A0302_Spintore".COut.Ax.MinusCheckNext AND "A0302_Spintore".COut.Vrt.Rest_CheckNext AND "A0302_Spintore".COut.Orz.Rest_CheckNext) OR ("A03_HMI".MB3.Button.A0302.SpintoreLong.OP.Work AND "A0302_Spintore".COut.Ax.PlusCheckNext AND "A0302_Spintore".COut.Vrt.Work_CheckNext AND "A0302_Spintore".COut.Orz.Work_CheckNext)) THEN
       #MB3_Decoder.OpEnabled := TRUE;
   END_IF;
   IF #_w1 AND (NOT "A0302_Spintore".COut.Ax.Standstill OR NOT "A0302_Spintore".COut.Vrt.Standstill OR NOT "A0302_Spintore".COut.Orz.Standstill) THEN
       #MB3_Decoder.OpRunning := TRUE;
   END_IF;
   IF #_w1 AND FALSE THEN #MB3_Decoder.OpDone := TRUE; END_IF;
END_REGION

REGION Network 26: MB3 Code 4012 - SPINTORE -AX
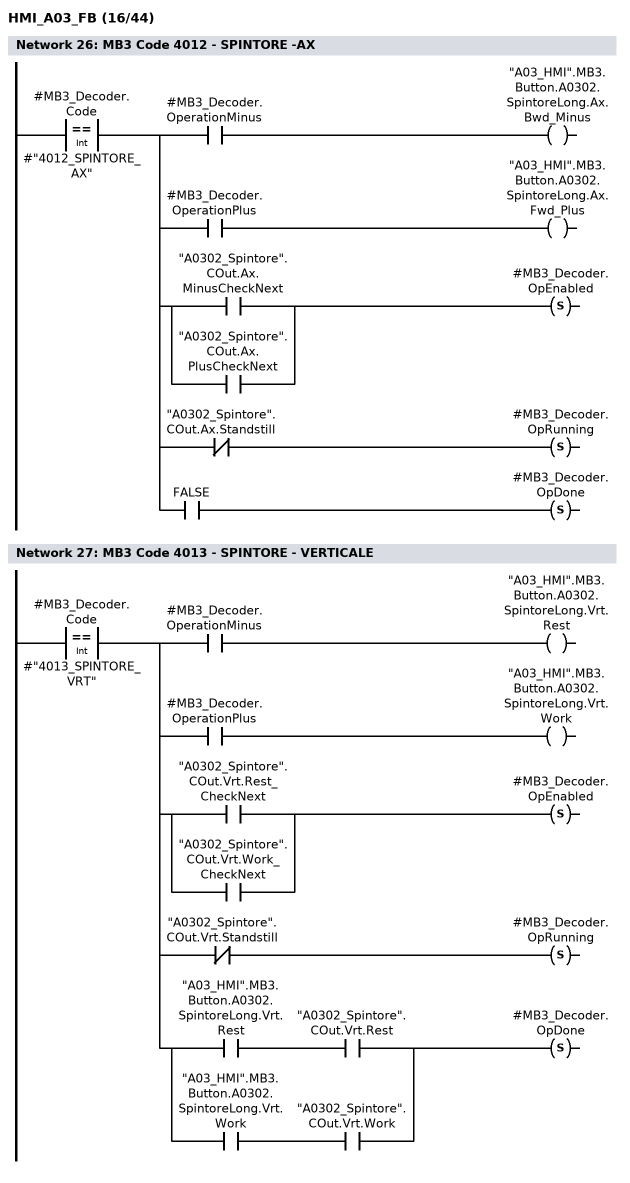
   RUNG wire#powerrail
      { S7_Templates := "SrcType := Int" } EQ_Contact(in1 := #MB3_Decoder.Code, in2 := #"4012_SPINTORE_AX")
      wire#w1
      Contact( #MB3_Decoder.OperationMinus )
      Coil( "A03_HMI".MB3.Button.A0302.SpintoreLong.Ax.Bwd_Minus )
   END_RUNG
   RUNG wire#w1
      Contact( #MB3_Decoder.OperationPlus )
      Coil( "A03_HMI".MB3.Button.A0302.SpintoreLong.Ax.Fwd_Plus )
   END_RUNG
   RUNG wire#w1
      Contact( "A0302_Spintore".COut.Ax.MinusCheckNext )
      wire#w2
      S_Coil( #MB3_Decoder.OpEnabled )
   END_RUNG
   RUNG wire#w1
      Contact( "A0302_Spintore".COut.Ax.PlusCheckNext )
   END_RUNG wire#w2
   RUNG wire#w1
      I_Contact( "A0302_Spintore".COut.Ax.Standstill )
      S_Coil( #MB3_Decoder.OpRunning )
   END_RUNG
   RUNG wire#w1
      Contact( FALSE )
      S_Coil( #MB3_Decoder.OpDone )
   END_RUNG
   // the same network as SCL:
   #_w1 := #MB3_Decoder.Code = #"4012_SPINTORE_AX";
   "A03_HMI".MB3.Button.A0302.SpintoreLong.Ax.Bwd_Minus := #_w1 AND #MB3_Decoder.OperationMinus;
   "A03_HMI".MB3.Button.A0302.SpintoreLong.Ax.Fwd_Plus := #_w1 AND #MB3_Decoder.OperationPlus;
   IF #_w1 AND ("A0302_Spintore".COut.Ax.MinusCheckNext OR "A0302_Spintore".COut.Ax.PlusCheckNext) THEN
       #MB3_Decoder.OpEnabled := TRUE;
   END_IF;
   IF #_w1 AND NOT "A0302_Spintore".COut.Ax.Standstill THEN #MB3_Decoder.OpRunning := TRUE; END_IF;
   IF #_w1 AND FALSE THEN #MB3_Decoder.OpDone := TRUE; END_IF;
END_REGION

REGION Network 27: MB3 Code 4013 - SPINTORE - VERTICALE
   RUNG wire#powerrail
      { S7_Templates := "SrcType := Int" } EQ_Contact(in1 := #MB3_Decoder.Code, in2 := #"4013_SPINTORE_VRT")
      wire#w1
      Contact( #MB3_Decoder.OperationMinus )
      Coil( "A03_HMI".MB3.Button.A0302.SpintoreLong.Vrt.Rest )
   END_RUNG
   RUNG wire#w1
      Contact( #MB3_Decoder.OperationPlus )
      Coil( "A03_HMI".MB3.Button.A0302.SpintoreLong.Vrt.Work )
   END_RUNG
   RUNG wire#w1
      Contact( "A0302_Spintore".COut.Vrt.Rest_CheckNext )
      wire#w2
      S_Coil( #MB3_Decoder.OpEnabled )
   END_RUNG
   RUNG wire#w1
      Contact( "A0302_Spintore".COut.Vrt.Work_CheckNext )
   END_RUNG wire#w2
   RUNG wire#w1
      I_Contact( "A0302_Spintore".COut.Vrt.Standstill )
      S_Coil( #MB3_Decoder.OpRunning )
   END_RUNG
   RUNG wire#w1
      Contact( "A03_HMI".MB3.Button.A0302.SpintoreLong.Vrt.Rest )
      Contact( "A0302_Spintore".COut.Vrt.Rest )
      wire#w3
      S_Coil( #MB3_Decoder.OpDone )
   END_RUNG
   RUNG wire#w1
      Contact( "A03_HMI".MB3.Button.A0302.SpintoreLong.Vrt.Work )
      Contact( "A0302_Spintore".COut.Vrt.Work )
   END_RUNG wire#w3
   // the same network as SCL:
   #_w1 := #MB3_Decoder.Code = #"4013_SPINTORE_VRT";
   "A03_HMI".MB3.Button.A0302.SpintoreLong.Vrt.Rest := #_w1 AND #MB3_Decoder.OperationMinus;
   "A03_HMI".MB3.Button.A0302.SpintoreLong.Vrt.Work := #_w1 AND #MB3_Decoder.OperationPlus;
   IF #_w1 AND ("A0302_Spintore".COut.Vrt.Rest_CheckNext OR "A0302_Spintore".COut.Vrt.Work_CheckNext) THEN
       #MB3_Decoder.OpEnabled := TRUE;
   END_IF;
   IF #_w1 AND NOT "A0302_Spintore".COut.Vrt.Standstill THEN #MB3_Decoder.OpRunning := TRUE; END_IF;
   IF #_w1 AND (("A03_HMI".MB3.Button.A0302.SpintoreLong.Vrt.Rest AND "A0302_Spintore".COut.Vrt.Rest) OR ("A03_HMI".MB3.Button.A0302.SpintoreLong.Vrt.Work AND "A0302_Spintore".COut.Vrt.Work)) THEN
       #MB3_Decoder.OpDone := TRUE;
   END_IF;
END_REGION

REGION Network 28: MB3 Code 4014 - SPINTORE - ORIZZONTALE
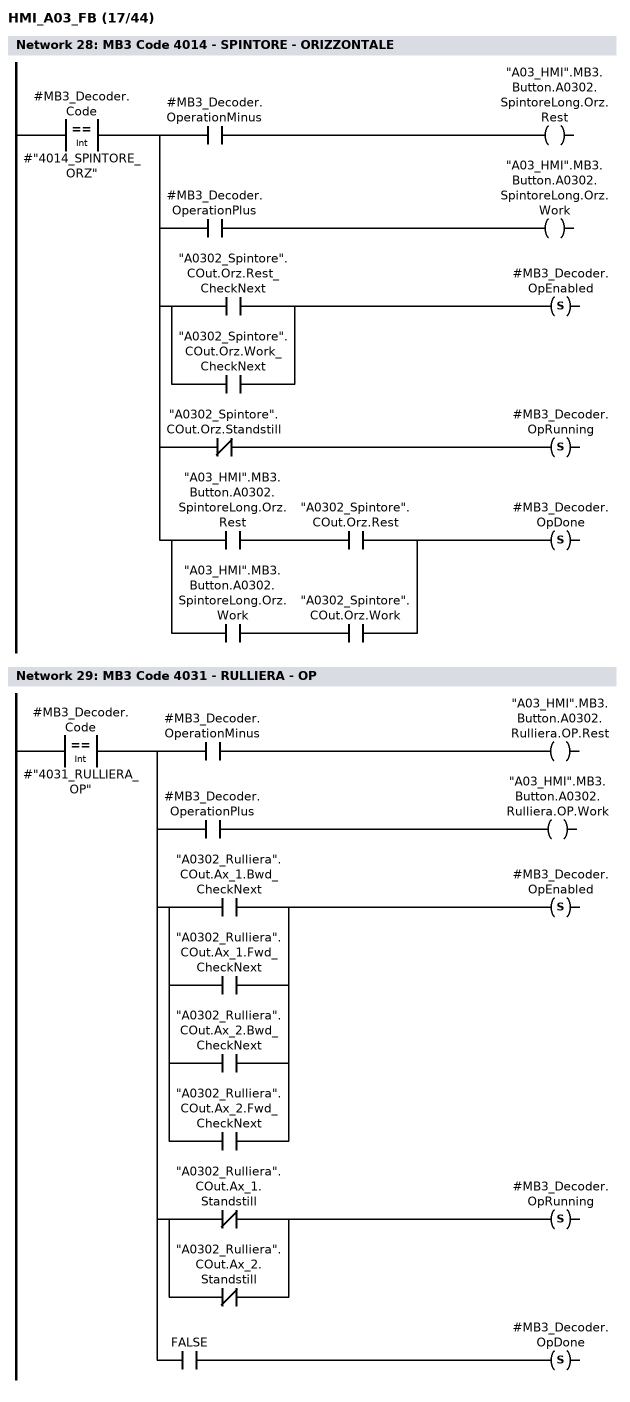
   RUNG wire#powerrail
      { S7_Templates := "SrcType := Int" } EQ_Contact(in1 := #MB3_Decoder.Code, in2 := #"4014_SPINTORE_ORZ")
      wire#w1
      Contact( #MB3_Decoder.OperationMinus )
      Coil( "A03_HMI".MB3.Button.A0302.SpintoreLong.Orz.Rest )
   END_RUNG
   RUNG wire#w1
      Contact( #MB3_Decoder.OperationPlus )
      Coil( "A03_HMI".MB3.Button.A0302.SpintoreLong.Orz.Work )
   END_RUNG
   RUNG wire#w1
      Contact( "A0302_Spintore".COut.Orz.Rest_CheckNext )
      wire#w2
      S_Coil( #MB3_Decoder.OpEnabled )
   END_RUNG
   RUNG wire#w1
      Contact( "A0302_Spintore".COut.Orz.Work_CheckNext )
   END_RUNG wire#w2
   RUNG wire#w1
      I_Contact( "A0302_Spintore".COut.Orz.Standstill )
      S_Coil( #MB3_Decoder.OpRunning )
   END_RUNG
   RUNG wire#w1
      Contact( "A03_HMI".MB3.Button.A0302.SpintoreLong.Orz.Rest )
      Contact( "A0302_Spintore".COut.Orz.Rest )
      wire#w3
      S_Coil( #MB3_Decoder.OpDone )
   END_RUNG
   RUNG wire#w1
      Contact( "A03_HMI".MB3.Button.A0302.SpintoreLong.Orz.Work )
      Contact( "A0302_Spintore".COut.Orz.Work )
   END_RUNG wire#w3
   // the same network as SCL:
   #_w1 := #MB3_Decoder.Code = #"4014_SPINTORE_ORZ";
   "A03_HMI".MB3.Button.A0302.SpintoreLong.Orz.Rest := #_w1 AND #MB3_Decoder.OperationMinus;
   "A03_HMI".MB3.Button.A0302.SpintoreLong.Orz.Work := #_w1 AND #MB3_Decoder.OperationPlus;
   IF #_w1 AND ("A0302_Spintore".COut.Orz.Rest_CheckNext OR "A0302_Spintore".COut.Orz.Work_CheckNext) THEN
       #MB3_Decoder.OpEnabled := TRUE;
   END_IF;
   IF #_w1 AND NOT "A0302_Spintore".COut.Orz.Standstill THEN #MB3_Decoder.OpRunning := TRUE; END_IF;
   IF #_w1 AND (("A03_HMI".MB3.Button.A0302.SpintoreLong.Orz.Rest AND "A0302_Spintore".COut.Orz.Rest) OR ("A03_HMI".MB3.Button.A0302.SpintoreLong.Orz.Work AND "A0302_Spintore".COut.Orz.Work)) THEN
       #MB3_Decoder.OpDone := TRUE;
   END_IF;
END_REGION

REGION Network 29: MB3 Code 4031 - RULLIERA - OP
   RUNG wire#powerrail
      { S7_Templates := "SrcType := Int" } EQ_Contact(in1 := #MB3_Decoder.Code, in2 := #"4031_RULLIERA_OP")
      wire#w1
      Contact( #MB3_Decoder.OperationMinus )
      Coil( "A03_HMI".MB3.Button.A0302.Rulliera.OP.Rest )
   END_RUNG
   RUNG wire#w1
      Contact( #MB3_Decoder.OperationPlus )
      Coil( "A03_HMI".MB3.Button.A0302.Rulliera.OP.Work )
   END_RUNG
   RUNG wire#w1
      Contact( "A0302_Rulliera".COut.Ax_1.Bwd_CheckNext )
      wire#w2
      S_Coil( #MB3_Decoder.OpEnabled )
   END_RUNG
   RUNG wire#w1
      Contact( "A0302_Rulliera".COut.Ax_1.Fwd_CheckNext )
   END_RUNG wire#w2
   RUNG wire#w1
      Contact( "A0302_Rulliera".COut.Ax_2.Bwd_CheckNext )
   END_RUNG wire#w2
   RUNG wire#w1
      Contact( "A0302_Rulliera".COut.Ax_2.Fwd_CheckNext )
   END_RUNG wire#w2
   RUNG wire#w1
      I_Contact( "A0302_Rulliera".COut.Ax_1.Standstill )
      wire#w3
      S_Coil( #MB3_Decoder.OpRunning )
   END_RUNG
   RUNG wire#w1
      I_Contact( "A0302_Rulliera".COut.Ax_2.Standstill )
   END_RUNG wire#w3
   RUNG wire#w1
      Contact( FALSE )
      S_Coil( #MB3_Decoder.OpDone )
   END_RUNG
   // the same network as SCL:
   #_w1 := #MB3_Decoder.Code = #"4031_RULLIERA_OP";
   "A03_HMI".MB3.Button.A0302.Rulliera.OP.Rest := #_w1 AND #MB3_Decoder.OperationMinus;
   "A03_HMI".MB3.Button.A0302.Rulliera.OP.Work := #_w1 AND #MB3_Decoder.OperationPlus;
   IF #_w1 AND ("A0302_Rulliera".COut.Ax_1.Bwd_CheckNext OR "A0302_Rulliera".COut.Ax_1.Fwd_CheckNext OR "A0302_Rulliera".COut.Ax_2.Bwd_CheckNext OR "A0302_Rulliera".COut.Ax_2.Fwd_CheckNext) THEN
       #MB3_Decoder.OpEnabled := TRUE;
   END_IF;
   IF #_w1 AND (NOT "A0302_Rulliera".COut.Ax_1.Standstill OR NOT "A0302_Rulliera".COut.Ax_2.Standstill) THEN
       #MB3_Decoder.OpRunning := TRUE;
   END_IF;
   IF #_w1 AND FALSE THEN #MB3_Decoder.OpDone := TRUE; END_IF;
END_REGION

REGION Network 30: MB3 Code 4032 - RULLIERA -AX
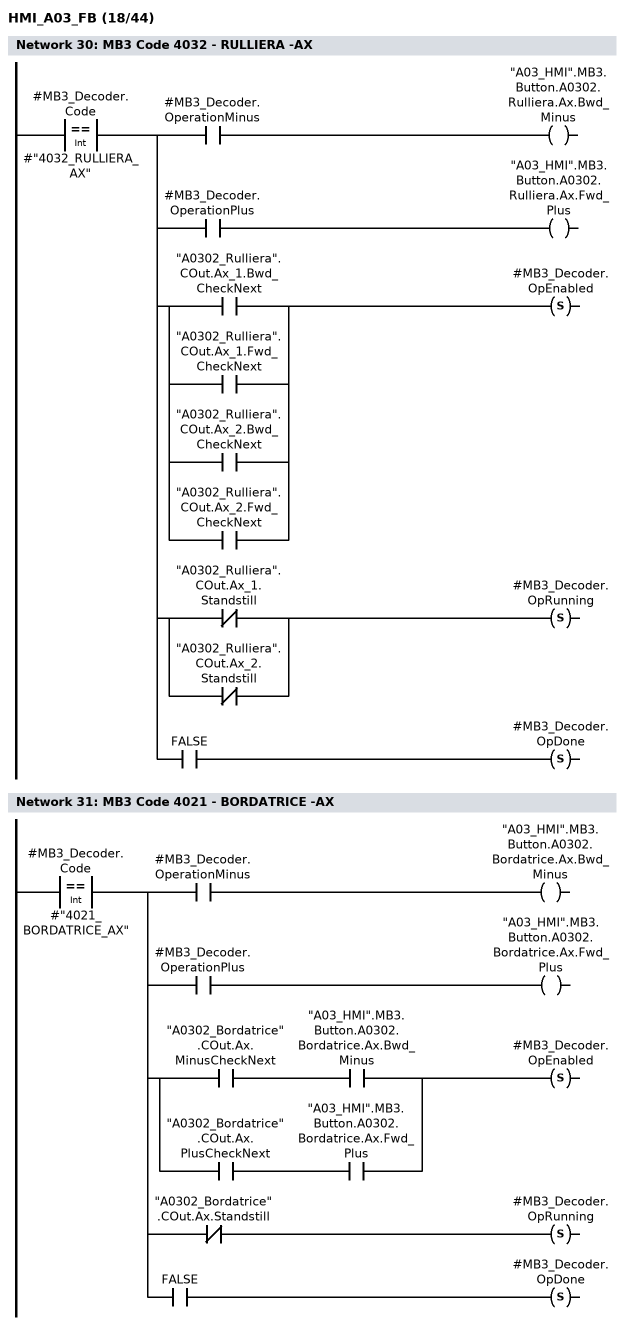
   RUNG wire#powerrail
      { S7_Templates := "SrcType := Int" } EQ_Contact(in1 := #MB3_Decoder.Code, in2 := #"4032_RULLIERA_AX")
      wire#w1
      Contact( #MB3_Decoder.OperationMinus )
      Coil( "A03_HMI".MB3.Button.A0302.Rulliera.Ax.Bwd_Minus )
   END_RUNG
   RUNG wire#w1
      Contact( #MB3_Decoder.OperationPlus )
      Coil( "A03_HMI".MB3.Button.A0302.Rulliera.Ax.Fwd_Plus )
   END_RUNG
   RUNG wire#w1
      Contact( "A0302_Rulliera".COut.Ax_1.Bwd_CheckNext )
      wire#w2
      S_Coil( #MB3_Decoder.OpEnabled )
   END_RUNG
   RUNG wire#w1
      Contact( "A0302_Rulliera".COut.Ax_1.Fwd_CheckNext )
   END_RUNG wire#w2
   RUNG wire#w1
      Contact( "A0302_Rulliera".COut.Ax_2.Bwd_CheckNext )
   END_RUNG wire#w2
   RUNG wire#w1
      Contact( "A0302_Rulliera".COut.Ax_2.Fwd_CheckNext )
   END_RUNG wire#w2
   RUNG wire#w1
      I_Contact( "A0302_Rulliera".COut.Ax_1.Standstill )
      wire#w3
      S_Coil( #MB3_Decoder.OpRunning )
   END_RUNG
   RUNG wire#w1
      I_Contact( "A0302_Rulliera".COut.Ax_2.Standstill )
   END_RUNG wire#w3
   RUNG wire#w1
      Contact( FALSE )
      S_Coil( #MB3_Decoder.OpDone )
   END_RUNG
   // the same network as SCL:
   #_w1 := #MB3_Decoder.Code = #"4032_RULLIERA_AX";
   "A03_HMI".MB3.Button.A0302.Rulliera.Ax.Bwd_Minus := #_w1 AND #MB3_Decoder.OperationMinus;
   "A03_HMI".MB3.Button.A0302.Rulliera.Ax.Fwd_Plus := #_w1 AND #MB3_Decoder.OperationPlus;
   IF #_w1 AND ("A0302_Rulliera".COut.Ax_1.Bwd_CheckNext OR "A0302_Rulliera".COut.Ax_1.Fwd_CheckNext OR "A0302_Rulliera".COut.Ax_2.Bwd_CheckNext OR "A0302_Rulliera".COut.Ax_2.Fwd_CheckNext) THEN
       #MB3_Decoder.OpEnabled := TRUE;
   END_IF;
   IF #_w1 AND (NOT "A0302_Rulliera".COut.Ax_1.Standstill OR NOT "A0302_Rulliera".COut.Ax_2.Standstill) THEN
       #MB3_Decoder.OpRunning := TRUE;
   END_IF;
   IF #_w1 AND FALSE THEN #MB3_Decoder.OpDone := TRUE; END_IF;
END_REGION

REGION Network 31: MB3 Code 4021 - BORDATRICE -AX
   RUNG wire#powerrail
      { S7_Templates := "SrcType := Int" } EQ_Contact(in1 := #MB3_Decoder.Code, in2 := #"4021_BORDATRICE_AX")
      wire#w1
      Contact( #MB3_Decoder.OperationMinus )
      Coil( "A03_HMI".MB3.Button.A0302.Bordatrice.Ax.Bwd_Minus )
   END_RUNG
   RUNG wire#w1
      Contact( #MB3_Decoder.OperationPlus )
      Coil( "A03_HMI".MB3.Button.A0302.Bordatrice.Ax.Fwd_Plus )
   END_RUNG
   RUNG wire#w1
      Contact( "A0302_Bordatrice".COut.Ax.MinusCheckNext )
      Contact( "A03_HMI".MB3.Button.A0302.Bordatrice.Ax.Bwd_Minus )
      wire#w2
      S_Coil( #MB3_Decoder.OpEnabled )
   END_RUNG
   RUNG wire#w1
      Contact( "A0302_Bordatrice".COut.Ax.PlusCheckNext )
      Contact( "A03_HMI".MB3.Button.A0302.Bordatrice.Ax.Fwd_Plus )
   END_RUNG wire#w2
   RUNG wire#w1
      I_Contact( "A0302_Bordatrice".COut.Ax.Standstill )
      S_Coil( #MB3_Decoder.OpRunning )
   END_RUNG
   RUNG wire#w1
      Contact( FALSE )
      S_Coil( #MB3_Decoder.OpDone )
   END_RUNG
   // the same network as SCL:
   #_w1 := #MB3_Decoder.Code = #"4021_BORDATRICE_AX";
   "A03_HMI".MB3.Button.A0302.Bordatrice.Ax.Bwd_Minus := #_w1 AND #MB3_Decoder.OperationMinus;
   "A03_HMI".MB3.Button.A0302.Bordatrice.Ax.Fwd_Plus := #_w1 AND #MB3_Decoder.OperationPlus;
   IF #_w1 AND (("A0302_Bordatrice".COut.Ax.MinusCheckNext AND "A03_HMI".MB3.Button.A0302.Bordatrice.Ax.Bwd_Minus) OR ("A0302_Bordatrice".COut.Ax.PlusCheckNext AND "A03_HMI".MB3.Button.A0302.Bordatrice.Ax.Fwd_Plus)) THEN
       #MB3_Decoder.OpEnabled := TRUE;
   END_IF;
   IF #_w1 AND NOT "A0302_Bordatrice".COut.Ax.Standstill THEN #MB3_Decoder.OpRunning := TRUE; END_IF;
   IF #_w1 AND FALSE THEN #MB3_Decoder.OpDone := TRUE; END_IF;
END_REGION

REGION Network 32: MB3 Code 4033 - REGOLAZ. BORDATRICE - CASSETTA
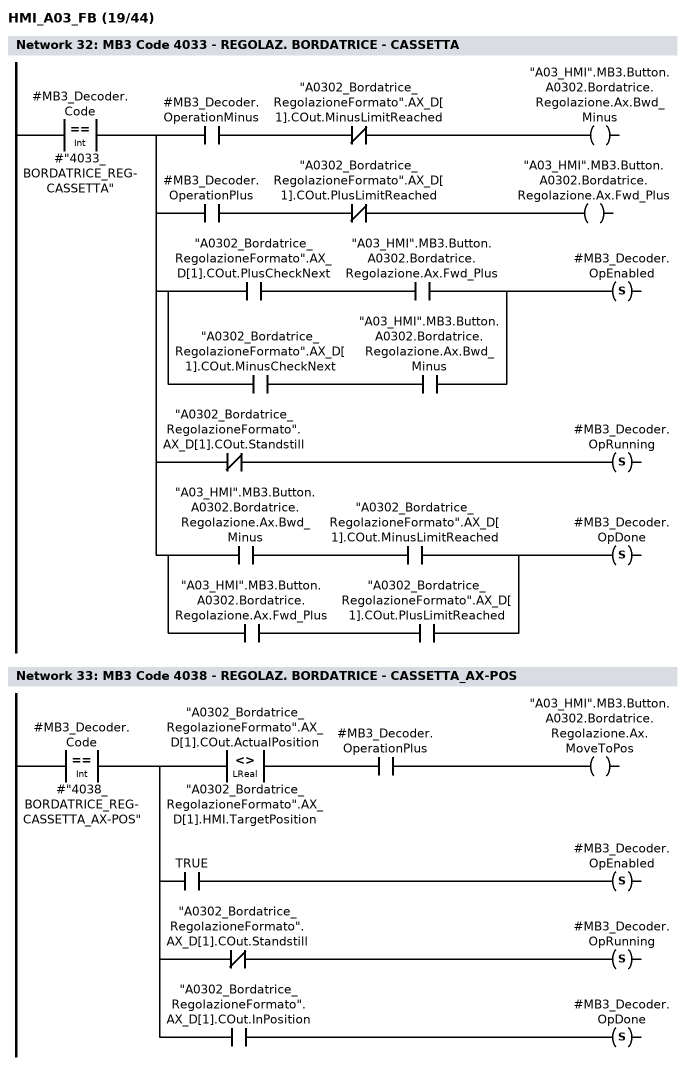
   RUNG wire#powerrail
      { S7_Templates := "SrcType := Int" } EQ_Contact(in1 := #MB3_Decoder.Code, in2 := #"4033_BORDATRICE_REG-CASSETTA")
      wire#w1
      Contact( #MB3_Decoder.OperationMinus )
      I_Contact( "A0302_Bordatrice_RegolazioneFormato".AX_D[1].COut.MinusLimitReached )
      Coil( "A03_HMI".MB3.Button.A0302.Bordatrice.Regolazione.Ax.Bwd_Minus )
   END_RUNG
   RUNG wire#w1
      Contact( #MB3_Decoder.OperationPlus )
      I_Contact( "A0302_Bordatrice_RegolazioneFormato".AX_D[1].COut.PlusLimitReached )
      Coil( "A03_HMI".MB3.Button.A0302.Bordatrice.Regolazione.Ax.Fwd_Plus )
   END_RUNG
   RUNG wire#w1
      Contact( "A0302_Bordatrice_RegolazioneFormato".AX_D[1].COut.PlusCheckNext )
      Contact( "A03_HMI".MB3.Button.A0302.Bordatrice.Regolazione.Ax.Fwd_Plus )
      wire#w2
      S_Coil( #MB3_Decoder.OpEnabled )
   END_RUNG
   RUNG wire#w1
      Contact( "A0302_Bordatrice_RegolazioneFormato".AX_D[1].COut.MinusCheckNext )
      Contact( "A03_HMI".MB3.Button.A0302.Bordatrice.Regolazione.Ax.Bwd_Minus )
   END_RUNG wire#w2
   RUNG wire#w1
      I_Contact( "A0302_Bordatrice_RegolazioneFormato".AX_D[1].COut.Standstill )
      S_Coil( #MB3_Decoder.OpRunning )
   END_RUNG
   RUNG wire#w1
      Contact( "A03_HMI".MB3.Button.A0302.Bordatrice.Regolazione.Ax.Bwd_Minus )
      Contact( "A0302_Bordatrice_RegolazioneFormato".AX_D[1].COut.MinusLimitReached )
      wire#w3
      S_Coil( #MB3_Decoder.OpDone )
   END_RUNG
   RUNG wire#w1
      Contact( "A03_HMI".MB3.Button.A0302.Bordatrice.Regolazione.Ax.Fwd_Plus )
      Contact( "A0302_Bordatrice_RegolazioneFormato".AX_D[1].COut.PlusLimitReached )
   END_RUNG wire#w3
   // the same network as SCL:
   #_w1 := #MB3_Decoder.Code = #"4033_BORDATRICE_REG-CASSETTA";
   "A03_HMI".MB3.Button.A0302.Bordatrice.Regolazione.Ax.Bwd_Minus := #_w1 AND #MB3_Decoder.OperationMinus AND NOT "A0302_Bordatrice_RegolazioneFormato".AX_D[1].COut.MinusLimitReached;
   "A03_HMI".MB3.Button.A0302.Bordatrice.Regolazione.Ax.Fwd_Plus := #_w1 AND #MB3_Decoder.OperationPlus AND NOT "A0302_Bordatrice_RegolazioneFormato".AX_D[1].COut.PlusLimitReached;
   IF #_w1 AND (("A0302_Bordatrice_RegolazioneFormato".AX_D[1].COut.PlusCheckNext AND "A03_HMI".MB3.Button.A0302.Bordatrice.Regolazione.Ax.Fwd_Plus) OR ("A0302_Bordatrice_RegolazioneFormato".AX_D[1].COut.MinusCheckNext AND "A03_HMI".MB3.Button.A0302.Bordatrice.Regolazione.Ax.Bwd_Minus)) THEN
       #MB3_Decoder.OpEnabled := TRUE;
   END_IF;
   IF #_w1 AND NOT "A0302_Bordatrice_RegolazioneFormato".AX_D[1].COut.Standstill THEN
       #MB3_Decoder.OpRunning := TRUE;
   END_IF;
   IF #_w1 AND (("A03_HMI".MB3.Button.A0302.Bordatrice.Regolazione.Ax.Bwd_Minus AND "A0302_Bordatrice_RegolazioneFormato".AX_D[1].COut.MinusLimitReached) OR ("A03_HMI".MB3.Button.A0302.Bordatrice.Regolazione.Ax.Fwd_Plus AND "A0302_Bordatrice_RegolazioneFormato".AX_D[1].COut.PlusLimitReached)) THEN
       #MB3_Decoder.OpDone := TRUE;
   END_IF;
END_REGION

REGION Network 33: MB3 Code 4038 - REGOLAZ. BORDATRICE - CASSETTA_AX-POS
   RUNG wire#powerrail
      { S7_Templates := "SrcType := Int" } EQ_Contact(in1 := #MB3_Decoder.Code, in2 := #"4038_BORDATRICE_REG-CASSETTA_AX-POS")
      wire#w1
      { S7_Templates := "SrcType := LReal" } NE_Contact(in1 := "A0302_Bordatrice_RegolazioneFormato".AX_D[1].COut.ActualPosition, in2 := "A0302_Bordatrice_RegolazioneFormato".AX_D[1].HMI.TargetPosition)
      Contact( #MB3_Decoder.OperationPlus )
      Coil( "A03_HMI".MB3.Button.A0302.Bordatrice.Regolazione.Ax.MoveToPos )
   END_RUNG
   RUNG wire#w1
      Contact( TRUE )
      S_Coil( #MB3_Decoder.OpEnabled )
   END_RUNG
   RUNG wire#w1
      I_Contact( "A0302_Bordatrice_RegolazioneFormato".AX_D[1].COut.Standstill )
      S_Coil( #MB3_Decoder.OpRunning )
   END_RUNG
   RUNG wire#w1
      Contact( "A0302_Bordatrice_RegolazioneFormato".AX_D[1].COut.InPosition )
      S_Coil( #MB3_Decoder.OpDone )
   END_RUNG
   // the same network as SCL:
   #_w1 := #MB3_Decoder.Code = #"4038_BORDATRICE_REG-CASSETTA_AX-POS";
   "A03_HMI".MB3.Button.A0302.Bordatrice.Regolazione.Ax.MoveToPos := #_w1 AND ("A0302_Bordatrice_RegolazioneFormato".AX_D[1].COut.ActualPosition <> "A0302_Bordatrice_RegolazioneFormato".AX_D[1].HMI.TargetPosition) AND #MB3_Decoder.OperationPlus;
   IF #_w1 AND TRUE THEN #MB3_Decoder.OpEnabled := TRUE; END_IF;
   IF #_w1 AND NOT "A0302_Bordatrice_RegolazioneFormato".AX_D[1].COut.Standstill THEN
       #MB3_Decoder.OpRunning := TRUE;
   END_IF;
   IF #_w1 AND "A0302_Bordatrice_RegolazioneFormato".AX_D[1].COut.InPosition THEN
       #MB3_Decoder.OpDone := TRUE;
   END_IF;
END_REGION

REGION Network 34: MB3 Code 4034 - REGOLAZ. BORDATRICE - PASSAGGIO 01 - COMBO
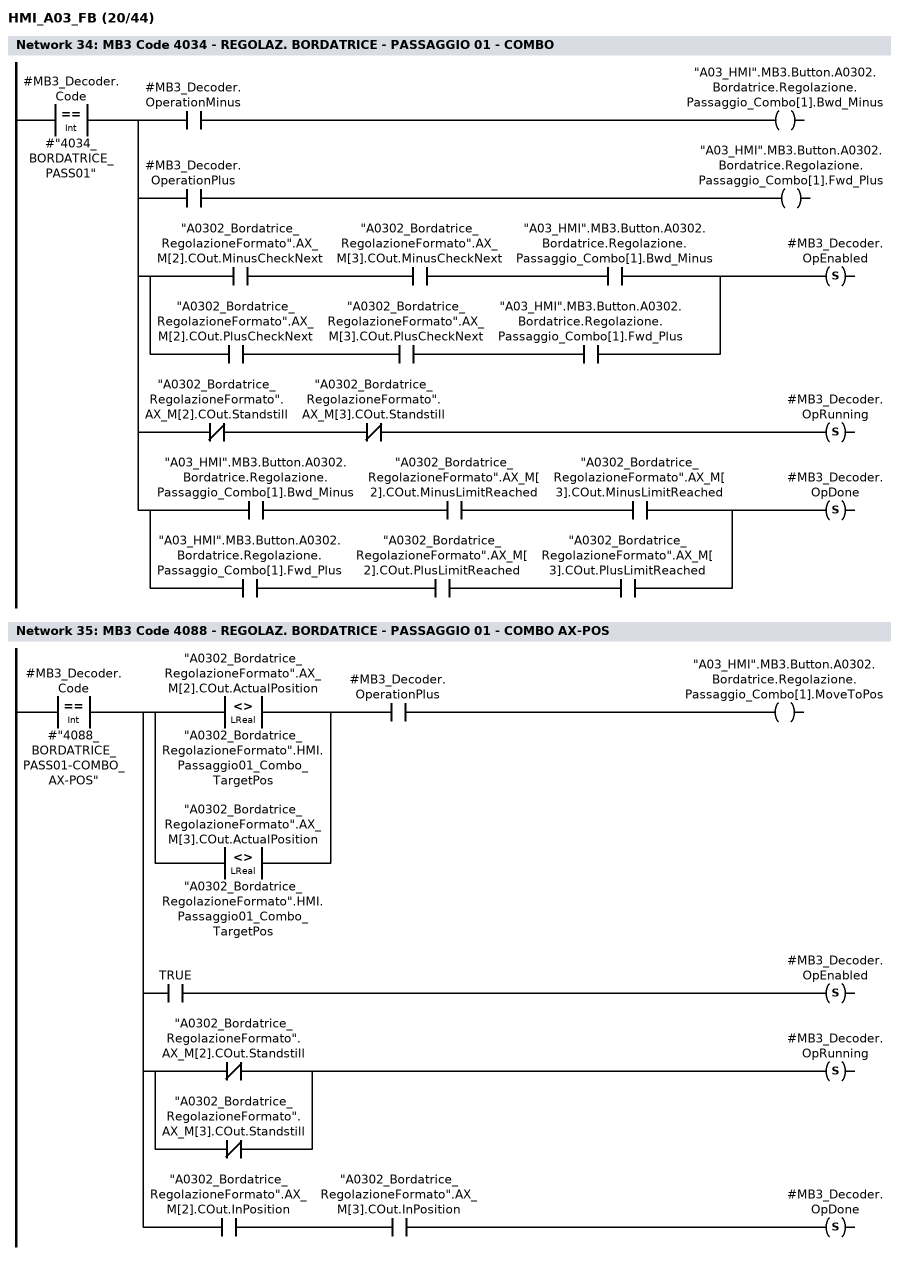
   RUNG wire#powerrail
      { S7_Templates := "SrcType := Int" } EQ_Contact(in1 := #MB3_Decoder.Code, in2 := #"4034_BORDATRICE_PASS01")
      wire#w1
      Contact( #MB3_Decoder.OperationMinus )
      Coil( "A03_HMI".MB3.Button.A0302.Bordatrice.Regolazione.Passaggio_Combo[1].Bwd_Minus )
   END_RUNG
   RUNG wire#w1
      Contact( #MB3_Decoder.OperationPlus )
      Coil( "A03_HMI".MB3.Button.A0302.Bordatrice.Regolazione.Passaggio_Combo[1].Fwd_Plus )
   END_RUNG
   RUNG wire#w1
      Contact( "A0302_Bordatrice_RegolazioneFormato".AX_M[2].COut.MinusCheckNext )
      Contact( "A0302_Bordatrice_RegolazioneFormato".AX_M[3].COut.MinusCheckNext )
      Contact( "A03_HMI".MB3.Button.A0302.Bordatrice.Regolazione.Passaggio_Combo[1].Bwd_Minus )
      wire#w2
      S_Coil( #MB3_Decoder.OpEnabled )
   END_RUNG
   RUNG wire#w1
      Contact( "A0302_Bordatrice_RegolazioneFormato".AX_M[2].COut.PlusCheckNext )
      Contact( "A0302_Bordatrice_RegolazioneFormato".AX_M[3].COut.PlusCheckNext )
      Contact( "A03_HMI".MB3.Button.A0302.Bordatrice.Regolazione.Passaggio_Combo[1].Fwd_Plus )
   END_RUNG wire#w2
   RUNG wire#w1
      I_Contact( "A0302_Bordatrice_RegolazioneFormato".AX_M[2].COut.Standstill )
      I_Contact( "A0302_Bordatrice_RegolazioneFormato".AX_M[3].COut.Standstill )
      S_Coil( #MB3_Decoder.OpRunning )
   END_RUNG
   RUNG wire#w1
      Contact( "A03_HMI".MB3.Button.A0302.Bordatrice.Regolazione.Passaggio_Combo[1].Bwd_Minus )
      Contact( "A0302_Bordatrice_RegolazioneFormato".AX_M[2].COut.MinusLimitReached )
      Contact( "A0302_Bordatrice_RegolazioneFormato".AX_M[3].COut.MinusLimitReached )
      wire#w3
      S_Coil( #MB3_Decoder.OpDone )
   END_RUNG
   RUNG wire#w1
      Contact( "A03_HMI".MB3.Button.A0302.Bordatrice.Regolazione.Passaggio_Combo[1].Fwd_Plus )
      Contact( "A0302_Bordatrice_RegolazioneFormato".AX_M[2].COut.PlusLimitReached )
      Contact( "A0302_Bordatrice_RegolazioneFormato".AX_M[3].COut.PlusLimitReached )
   END_RUNG wire#w3
   // the same network as SCL:
   #_w1 := #MB3_Decoder.Code = #"4034_BORDATRICE_PASS01";
   "A03_HMI".MB3.Button.A0302.Bordatrice.Regolazione.Passaggio_Combo[1].Bwd_Minus := #_w1 AND #MB3_Decoder.OperationMinus;
   "A03_HMI".MB3.Button.A0302.Bordatrice.Regolazione.Passaggio_Combo[1].Fwd_Plus := #_w1 AND #MB3_Decoder.OperationPlus;
   IF #_w1 AND (("A0302_Bordatrice_RegolazioneFormato".AX_M[2].COut.MinusCheckNext AND "A0302_Bordatrice_RegolazioneFormato".AX_M[3].COut.MinusCheckNext AND "A03_HMI".MB3.Button.A0302.Bordatrice.Regolazione.Passaggio_Combo[1].Bwd_Minus) OR ("A0302_Bordatrice_RegolazioneFormato".AX_M[2].COut.PlusCheckNext AND "A0302_Bordatrice_RegolazioneFormato".AX_M[3].COut.PlusCheckNext AND "A03_HMI".MB3.Button.A0302.Bordatrice.Regolazione.Passaggio_Combo[1].Fwd_Plus)) THEN
       #MB3_Decoder.OpEnabled := TRUE;
   END_IF;
   IF #_w1 AND NOT "A0302_Bordatrice_RegolazioneFormato".AX_M[2].COut.Standstill AND NOT "A0302_Bordatrice_RegolazioneFormato".AX_M[3].COut.Standstill THEN
       #MB3_Decoder.OpRunning := TRUE;
   END_IF;
   IF #_w1 AND (("A03_HMI".MB3.Button.A0302.Bordatrice.Regolazione.Passaggio_Combo[1].Bwd_Minus AND "A0302_Bordatrice_RegolazioneFormato".AX_M[2].COut.MinusLimitReached AND "A0302_Bordatrice_RegolazioneFormato".AX_M[3].COut.MinusLimitReached) OR ("A03_HMI".MB3.Button.A0302.Bordatrice.Regolazione.Passaggio_Combo[1].Fwd_Plus AND "A0302_Bordatrice_RegolazioneFormato".AX_M[2].COut.PlusLimitReached AND "A0302_Bordatrice_RegolazioneFormato".AX_M[3].COut.PlusLimitReached)) THEN
       #MB3_Decoder.OpDone := TRUE;
   END_IF;
END_REGION

REGION Network 35: MB3 Code 4088 - REGOLAZ. BORDATRICE - PASSAGGIO 01 - COMBO AX-POS
   RUNG wire#powerrail
      { S7_Templates := "SrcType := Int" } EQ_Contact(in1 := #MB3_Decoder.Code, in2 := #"4088_BORDATRICE_PASS01-COMBO_AX-POS")
      wire#w1
      { S7_Templates := "SrcType := LReal" } NE_Contact(in1 := "A0302_Bordatrice_RegolazioneFormato".AX_M[2].COut.ActualPosition, in2 := "A0302_Bordatrice_RegolazioneFormato".HMI.Passaggio01_Combo_TargetPos)
      wire#w2
      Contact( #MB3_Decoder.OperationPlus )
      Coil( "A03_HMI".MB3.Button.A0302.Bordatrice.Regolazione.Passaggio_Combo[1].MoveToPos )
   END_RUNG
   RUNG wire#w1
      { S7_Templates := "SrcType := LReal" } NE_Contact(in1 := "A0302_Bordatrice_RegolazioneFormato".AX_M[3].COut.ActualPosition, in2 := "A0302_Bordatrice_RegolazioneFormato".HMI.Passaggio01_Combo_TargetPos)
   END_RUNG wire#w2
   RUNG wire#w1
      Contact( TRUE )
      S_Coil( #MB3_Decoder.OpEnabled )
   END_RUNG
   RUNG wire#w1
      I_Contact( "A0302_Bordatrice_RegolazioneFormato".AX_M[2].COut.Standstill )
      wire#w3
      S_Coil( #MB3_Decoder.OpRunning )
   END_RUNG
   RUNG wire#w1
      I_Contact( "A0302_Bordatrice_RegolazioneFormato".AX_M[3].COut.Standstill )
   END_RUNG wire#w3
   RUNG wire#w1
      Contact( "A0302_Bordatrice_RegolazioneFormato".AX_M[2].COut.InPosition )
      Contact( "A0302_Bordatrice_RegolazioneFormato".AX_M[3].COut.InPosition )
      S_Coil( #MB3_Decoder.OpDone )
   END_RUNG
   // the same network as SCL:
   #_w1 := #MB3_Decoder.Code = #"4088_BORDATRICE_PASS01-COMBO_AX-POS";
   "A03_HMI".MB3.Button.A0302.Bordatrice.Regolazione.Passaggio_Combo[1].MoveToPos := #_w1 AND (("A0302_Bordatrice_RegolazioneFormato".AX_M[2].COut.ActualPosition <> "A0302_Bordatrice_RegolazioneFormato".HMI.Passaggio01_Combo_TargetPos) OR ("A0302_Bordatrice_RegolazioneFormato".AX_M[3].COut.ActualPosition <> "A0302_Bordatrice_RegolazioneFormato".HMI.Passaggio01_Combo_TargetPos)) AND #MB3_Decoder.OperationPlus;
   IF #_w1 AND TRUE THEN #MB3_Decoder.OpEnabled := TRUE; END_IF;
   IF #_w1 AND (NOT "A0302_Bordatrice_RegolazioneFormato".AX_M[2].COut.Standstill OR NOT "A0302_Bordatrice_RegolazioneFormato".AX_M[3].COut.Standstill) THEN
       #MB3_Decoder.OpRunning := TRUE;
   END_IF;
   IF #_w1 AND "A0302_Bordatrice_RegolazioneFormato".AX_M[2].COut.InPosition AND "A0302_Bordatrice_RegolazioneFormato".AX_M[3].COut.InPosition THEN
       #MB3_Decoder.OpDone := TRUE;
   END_IF;
END_REGION

REGION Network 36: MB3 Code 4080 - REGOLAZ. BORDATRICE - PASSAGGIO 01 - LATO-OP
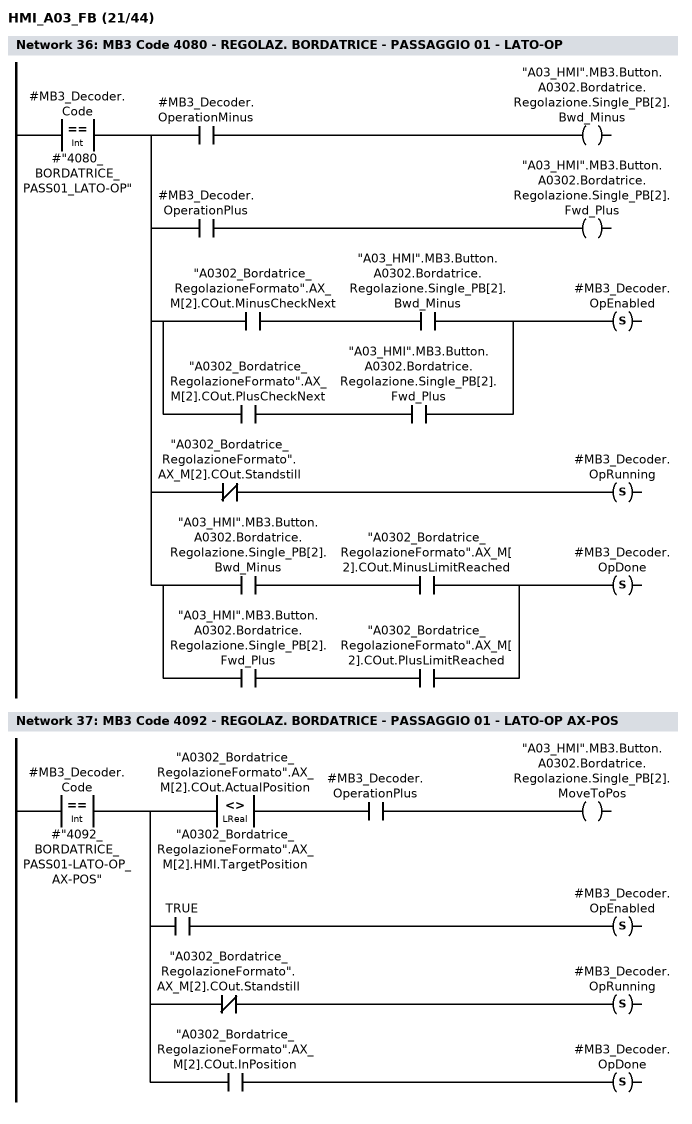
   RUNG wire#powerrail
      { S7_Templates := "SrcType := Int" } EQ_Contact(in1 := #MB3_Decoder.Code, in2 := #"4080_BORDATRICE_PASS01_LATO-OP")
      wire#w1
      Contact( #MB3_Decoder.OperationMinus )
      Coil( "A03_HMI".MB3.Button.A0302.Bordatrice.Regolazione.Single_PB[2].Bwd_Minus )
   END_RUNG
   RUNG wire#w1
      Contact( #MB3_Decoder.OperationPlus )
      Coil( "A03_HMI".MB3.Button.A0302.Bordatrice.Regolazione.Single_PB[2].Fwd_Plus )
   END_RUNG
   RUNG wire#w1
      Contact( "A0302_Bordatrice_RegolazioneFormato".AX_M[2].COut.MinusCheckNext )
      Contact( "A03_HMI".MB3.Button.A0302.Bordatrice.Regolazione.Single_PB[2].Bwd_Minus )
      wire#w2
      S_Coil( #MB3_Decoder.OpEnabled )
   END_RUNG
   RUNG wire#w1
      Contact( "A0302_Bordatrice_RegolazioneFormato".AX_M[2].COut.PlusCheckNext )
      Contact( "A03_HMI".MB3.Button.A0302.Bordatrice.Regolazione.Single_PB[2].Fwd_Plus )
   END_RUNG wire#w2
   RUNG wire#w1
      I_Contact( "A0302_Bordatrice_RegolazioneFormato".AX_M[2].COut.Standstill )
      S_Coil( #MB3_Decoder.OpRunning )
   END_RUNG
   RUNG wire#w1
      Contact( "A03_HMI".MB3.Button.A0302.Bordatrice.Regolazione.Single_PB[2].Bwd_Minus )
      Contact( "A0302_Bordatrice_RegolazioneFormato".AX_M[2].COut.MinusLimitReached )
      wire#w3
      S_Coil( #MB3_Decoder.OpDone )
   END_RUNG
   RUNG wire#w1
      Contact( "A03_HMI".MB3.Button.A0302.Bordatrice.Regolazione.Single_PB[2].Fwd_Plus )
      Contact( "A0302_Bordatrice_RegolazioneFormato".AX_M[2].COut.PlusLimitReached )
   END_RUNG wire#w3
   // the same network as SCL:
   #_w1 := #MB3_Decoder.Code = #"4080_BORDATRICE_PASS01_LATO-OP";
   "A03_HMI".MB3.Button.A0302.Bordatrice.Regolazione.Single_PB[2].Bwd_Minus := #_w1 AND #MB3_Decoder.OperationMinus;
   "A03_HMI".MB3.Button.A0302.Bordatrice.Regolazione.Single_PB[2].Fwd_Plus := #_w1 AND #MB3_Decoder.OperationPlus;
   IF #_w1 AND (("A0302_Bordatrice_RegolazioneFormato".AX_M[2].COut.MinusCheckNext AND "A03_HMI".MB3.Button.A0302.Bordatrice.Regolazione.Single_PB[2].Bwd_Minus) OR ("A0302_Bordatrice_RegolazioneFormato".AX_M[2].COut.PlusCheckNext AND "A03_HMI".MB3.Button.A0302.Bordatrice.Regolazione.Single_PB[2].Fwd_Plus)) THEN
       #MB3_Decoder.OpEnabled := TRUE;
   END_IF;
   IF #_w1 AND NOT "A0302_Bordatrice_RegolazioneFormato".AX_M[2].COut.Standstill THEN
       #MB3_Decoder.OpRunning := TRUE;
   END_IF;
   IF #_w1 AND (("A03_HMI".MB3.Button.A0302.Bordatrice.Regolazione.Single_PB[2].Bwd_Minus AND "A0302_Bordatrice_RegolazioneFormato".AX_M[2].COut.MinusLimitReached) OR ("A03_HMI".MB3.Button.A0302.Bordatrice.Regolazione.Single_PB[2].Fwd_Plus AND "A0302_Bordatrice_RegolazioneFormato".AX_M[2].COut.PlusLimitReached)) THEN
       #MB3_Decoder.OpDone := TRUE;
   END_IF;
END_REGION

REGION Network 37: MB3 Code 4092 - REGOLAZ. BORDATRICE - PASSAGGIO 01 - LATO-OP AX-POS
   RUNG wire#powerrail
      { S7_Templates := "SrcType := Int" } EQ_Contact(in1 := #MB3_Decoder.Code, in2 := #"4092_BORDATRICE_PASS01-LATO-OP_AX-POS")
      wire#w1
      { S7_Templates := "SrcType := LReal" } NE_Contact(in1 := "A0302_Bordatrice_RegolazioneFormato".AX_M[2].COut.ActualPosition, in2 := "A0302_Bordatrice_RegolazioneFormato".AX_M[2].HMI.TargetPosition)
      Contact( #MB3_Decoder.OperationPlus )
      Coil( "A03_HMI".MB3.Button.A0302.Bordatrice.Regolazione.Single_PB[2].MoveToPos )
   END_RUNG
   RUNG wire#w1
      Contact( TRUE )
      S_Coil( #MB3_Decoder.OpEnabled )
   END_RUNG
   RUNG wire#w1
      I_Contact( "A0302_Bordatrice_RegolazioneFormato".AX_M[2].COut.Standstill )
      S_Coil( #MB3_Decoder.OpRunning )
   END_RUNG
   RUNG wire#w1
      Contact( "A0302_Bordatrice_RegolazioneFormato".AX_M[2].COut.InPosition )
      S_Coil( #MB3_Decoder.OpDone )
   END_RUNG
   // the same network as SCL:
   #_w1 := #MB3_Decoder.Code = #"4092_BORDATRICE_PASS01-LATO-OP_AX-POS";
   "A03_HMI".MB3.Button.A0302.Bordatrice.Regolazione.Single_PB[2].MoveToPos := #_w1 AND ("A0302_Bordatrice_RegolazioneFormato".AX_M[2].COut.ActualPosition <> "A0302_Bordatrice_RegolazioneFormato".AX_M[2].HMI.TargetPosition) AND #MB3_Decoder.OperationPlus;
   IF #_w1 AND TRUE THEN #MB3_Decoder.OpEnabled := TRUE; END_IF;
   IF #_w1 AND NOT "A0302_Bordatrice_RegolazioneFormato".AX_M[2].COut.Standstill THEN
       #MB3_Decoder.OpRunning := TRUE;
   END_IF;
   IF #_w1 AND "A0302_Bordatrice_RegolazioneFormato".AX_M[2].COut.InPosition THEN
       #MB3_Decoder.OpDone := TRUE;
   END_IF;
END_REGION

REGION Network 38: MB3 Code 4081 - REGOLAZ. BORDATRICE - PASSAGGIO 01 - LATO-MOT
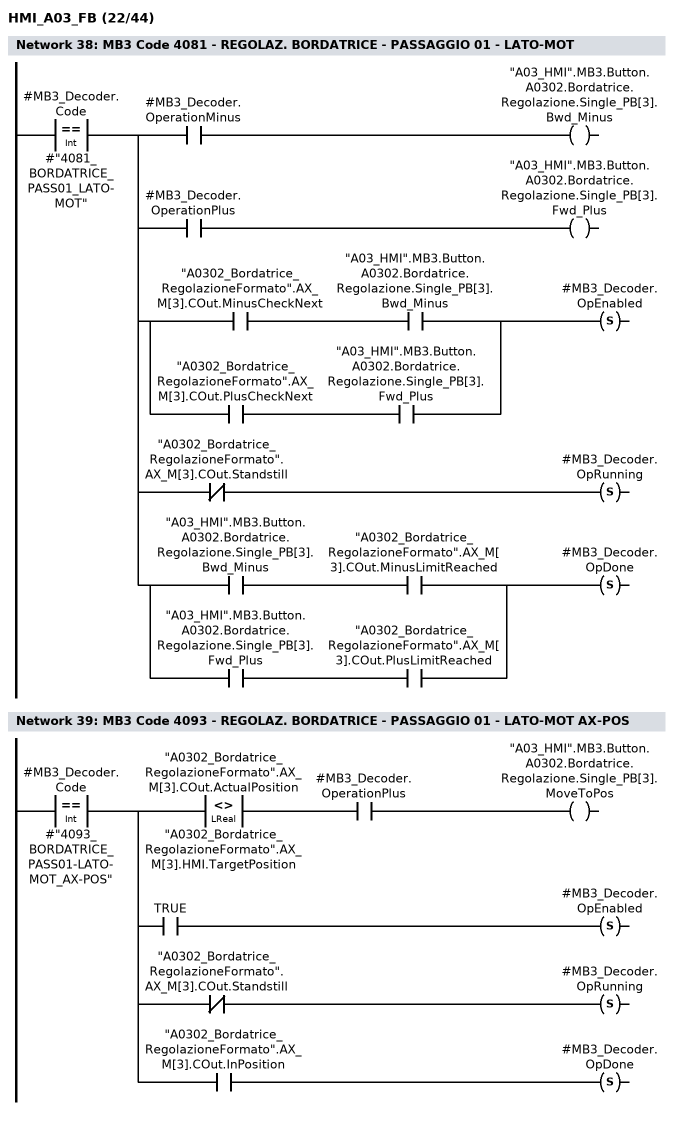
   RUNG wire#powerrail
      { S7_Templates := "SrcType := Int" } EQ_Contact(in1 := #MB3_Decoder.Code, in2 := #"4081_BORDATRICE_PASS01_LATO-MOT")
      wire#w1
      Contact( #MB3_Decoder.OperationMinus )
      Coil( "A03_HMI".MB3.Button.A0302.Bordatrice.Regolazione.Single_PB[3].Bwd_Minus )
   END_RUNG
   RUNG wire#w1
      Contact( #MB3_Decoder.OperationPlus )
      Coil( "A03_HMI".MB3.Button.A0302.Bordatrice.Regolazione.Single_PB[3].Fwd_Plus )
   END_RUNG
   RUNG wire#w1
      Contact( "A0302_Bordatrice_RegolazioneFormato".AX_M[3].COut.MinusCheckNext )
      Contact( "A03_HMI".MB3.Button.A0302.Bordatrice.Regolazione.Single_PB[3].Bwd_Minus )
      wire#w2
      S_Coil( #MB3_Decoder.OpEnabled )
   END_RUNG
   RUNG wire#w1
      Contact( "A0302_Bordatrice_RegolazioneFormato".AX_M[3].COut.PlusCheckNext )
      Contact( "A03_HMI".MB3.Button.A0302.Bordatrice.Regolazione.Single_PB[3].Fwd_Plus )
   END_RUNG wire#w2
   RUNG wire#w1
      I_Contact( "A0302_Bordatrice_RegolazioneFormato".AX_M[3].COut.Standstill )
      S_Coil( #MB3_Decoder.OpRunning )
   END_RUNG
   RUNG wire#w1
      Contact( "A03_HMI".MB3.Button.A0302.Bordatrice.Regolazione.Single_PB[3].Bwd_Minus )
      Contact( "A0302_Bordatrice_RegolazioneFormato".AX_M[3].COut.MinusLimitReached )
      wire#w3
      S_Coil( #MB3_Decoder.OpDone )
   END_RUNG
   RUNG wire#w1
      Contact( "A03_HMI".MB3.Button.A0302.Bordatrice.Regolazione.Single_PB[3].Fwd_Plus )
      Contact( "A0302_Bordatrice_RegolazioneFormato".AX_M[3].COut.PlusLimitReached )
   END_RUNG wire#w3
   // the same network as SCL:
   #_w1 := #MB3_Decoder.Code = #"4081_BORDATRICE_PASS01_LATO-MOT";
   "A03_HMI".MB3.Button.A0302.Bordatrice.Regolazione.Single_PB[3].Bwd_Minus := #_w1 AND #MB3_Decoder.OperationMinus;
   "A03_HMI".MB3.Button.A0302.Bordatrice.Regolazione.Single_PB[3].Fwd_Plus := #_w1 AND #MB3_Decoder.OperationPlus;
   IF #_w1 AND (("A0302_Bordatrice_RegolazioneFormato".AX_M[3].COut.MinusCheckNext AND "A03_HMI".MB3.Button.A0302.Bordatrice.Regolazione.Single_PB[3].Bwd_Minus) OR ("A0302_Bordatrice_RegolazioneFormato".AX_M[3].COut.PlusCheckNext AND "A03_HMI".MB3.Button.A0302.Bordatrice.Regolazione.Single_PB[3].Fwd_Plus)) THEN
       #MB3_Decoder.OpEnabled := TRUE;
   END_IF;
   IF #_w1 AND NOT "A0302_Bordatrice_RegolazioneFormato".AX_M[3].COut.Standstill THEN
       #MB3_Decoder.OpRunning := TRUE;
   END_IF;
   IF #_w1 AND (("A03_HMI".MB3.Button.A0302.Bordatrice.Regolazione.Single_PB[3].Bwd_Minus AND "A0302_Bordatrice_RegolazioneFormato".AX_M[3].COut.MinusLimitReached) OR ("A03_HMI".MB3.Button.A0302.Bordatrice.Regolazione.Single_PB[3].Fwd_Plus AND "A0302_Bordatrice_RegolazioneFormato".AX_M[3].COut.PlusLimitReached)) THEN
       #MB3_Decoder.OpDone := TRUE;
   END_IF;
END_REGION

REGION Network 39: MB3 Code 4093 - REGOLAZ. BORDATRICE - PASSAGGIO 01 - LATO-MOT AX-POS
   RUNG wire#powerrail
      { S7_Templates := "SrcType := Int" } EQ_Contact(in1 := #MB3_Decoder.Code, in2 := #"4093_BORDATRICE_PASS01-LATO-MOT_AX-POS")
      wire#w1
      { S7_Templates := "SrcType := LReal" } NE_Contact(in1 := "A0302_Bordatrice_RegolazioneFormato".AX_M[3].COut.ActualPosition, in2 := "A0302_Bordatrice_RegolazioneFormato".AX_M[3].HMI.TargetPosition)
      Contact( #MB3_Decoder.OperationPlus )
      Coil( "A03_HMI".MB3.Button.A0302.Bordatrice.Regolazione.Single_PB[3].MoveToPos )
   END_RUNG
   RUNG wire#w1
      Contact( TRUE )
      S_Coil( #MB3_Decoder.OpEnabled )
   END_RUNG
   RUNG wire#w1
      I_Contact( "A0302_Bordatrice_RegolazioneFormato".AX_M[3].COut.Standstill )
      S_Coil( #MB3_Decoder.OpRunning )
   END_RUNG
   RUNG wire#w1
      Contact( "A0302_Bordatrice_RegolazioneFormato".AX_M[3].COut.InPosition )
      S_Coil( #MB3_Decoder.OpDone )
   END_RUNG
   // the same network as SCL:
   #_w1 := #MB3_Decoder.Code = #"4093_BORDATRICE_PASS01-LATO-MOT_AX-POS";
   "A03_HMI".MB3.Button.A0302.Bordatrice.Regolazione.Single_PB[3].MoveToPos := #_w1 AND ("A0302_Bordatrice_RegolazioneFormato".AX_M[3].COut.ActualPosition <> "A0302_Bordatrice_RegolazioneFormato".AX_M[3].HMI.TargetPosition) AND #MB3_Decoder.OperationPlus;
   IF #_w1 AND TRUE THEN #MB3_Decoder.OpEnabled := TRUE; END_IF;
   IF #_w1 AND NOT "A0302_Bordatrice_RegolazioneFormato".AX_M[3].COut.Standstill THEN
       #MB3_Decoder.OpRunning := TRUE;
   END_IF;
   IF #_w1 AND "A0302_Bordatrice_RegolazioneFormato".AX_M[3].COut.InPosition THEN
       #MB3_Decoder.OpDone := TRUE;
   END_IF;
END_REGION

REGION Network 40: MB3 Code 4035 - REGOLAZ. BORDATRICE - PASSAGGIO 02 - COMBO
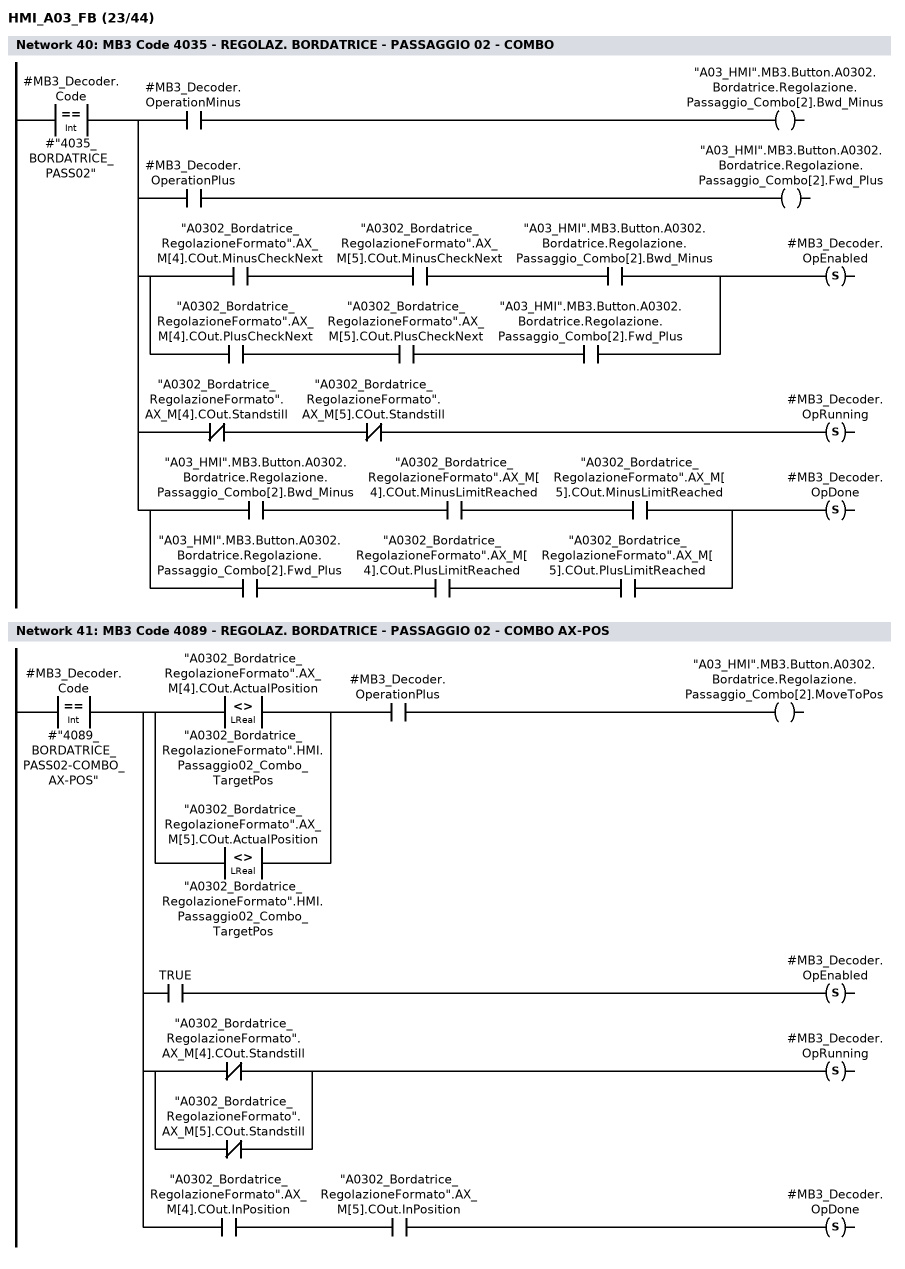
   RUNG wire#powerrail
      { S7_Templates := "SrcType := Int" } EQ_Contact(in1 := #MB3_Decoder.Code, in2 := #"4035_BORDATRICE_PASS02")
      wire#w1
      Contact( #MB3_Decoder.OperationMinus )
      Coil( "A03_HMI".MB3.Button.A0302.Bordatrice.Regolazione.Passaggio_Combo[2].Bwd_Minus )
   END_RUNG
   RUNG wire#w1
      Contact( #MB3_Decoder.OperationPlus )
      Coil( "A03_HMI".MB3.Button.A0302.Bordatrice.Regolazione.Passaggio_Combo[2].Fwd_Plus )
   END_RUNG
   RUNG wire#w1
      Contact( "A0302_Bordatrice_RegolazioneFormato".AX_M[4].COut.MinusCheckNext )
      Contact( "A0302_Bordatrice_RegolazioneFormato".AX_M[5].COut.MinusCheckNext )
      Contact( "A03_HMI".MB3.Button.A0302.Bordatrice.Regolazione.Passaggio_Combo[2].Bwd_Minus )
      wire#w2
      S_Coil( #MB3_Decoder.OpEnabled )
   END_RUNG
   RUNG wire#w1
      Contact( "A0302_Bordatrice_RegolazioneFormato".AX_M[4].COut.PlusCheckNext )
      Contact( "A0302_Bordatrice_RegolazioneFormato".AX_M[5].COut.PlusCheckNext )
      Contact( "A03_HMI".MB3.Button.A0302.Bordatrice.Regolazione.Passaggio_Combo[2].Fwd_Plus )
   END_RUNG wire#w2
   RUNG wire#w1
      I_Contact( "A0302_Bordatrice_RegolazioneFormato".AX_M[4].COut.Standstill )
      I_Contact( "A0302_Bordatrice_RegolazioneFormato".AX_M[5].COut.Standstill )
      S_Coil( #MB3_Decoder.OpRunning )
   END_RUNG
   RUNG wire#w1
      Contact( "A03_HMI".MB3.Button.A0302.Bordatrice.Regolazione.Passaggio_Combo[2].Bwd_Minus )
      Contact( "A0302_Bordatrice_RegolazioneFormato".AX_M[4].COut.MinusLimitReached )
      Contact( "A0302_Bordatrice_RegolazioneFormato".AX_M[5].COut.MinusLimitReached )
      wire#w3
      S_Coil( #MB3_Decoder.OpDone )
   END_RUNG
   RUNG wire#w1
      Contact( "A03_HMI".MB3.Button.A0302.Bordatrice.Regolazione.Passaggio_Combo[2].Fwd_Plus )
      Contact( "A0302_Bordatrice_RegolazioneFormato".AX_M[4].COut.PlusLimitReached )
      Contact( "A0302_Bordatrice_RegolazioneFormato".AX_M[5].COut.PlusLimitReached )
   END_RUNG wire#w3
   // the same network as SCL:
   #_w1 := #MB3_Decoder.Code = #"4035_BORDATRICE_PASS02";
   "A03_HMI".MB3.Button.A0302.Bordatrice.Regolazione.Passaggio_Combo[2].Bwd_Minus := #_w1 AND #MB3_Decoder.OperationMinus;
   "A03_HMI".MB3.Button.A0302.Bordatrice.Regolazione.Passaggio_Combo[2].Fwd_Plus := #_w1 AND #MB3_Decoder.OperationPlus;
   IF #_w1 AND (("A0302_Bordatrice_RegolazioneFormato".AX_M[4].COut.MinusCheckNext AND "A0302_Bordatrice_RegolazioneFormato".AX_M[5].COut.MinusCheckNext AND "A03_HMI".MB3.Button.A0302.Bordatrice.Regolazione.Passaggio_Combo[2].Bwd_Minus) OR ("A0302_Bordatrice_RegolazioneFormato".AX_M[4].COut.PlusCheckNext AND "A0302_Bordatrice_RegolazioneFormato".AX_M[5].COut.PlusCheckNext AND "A03_HMI".MB3.Button.A0302.Bordatrice.Regolazione.Passaggio_Combo[2].Fwd_Plus)) THEN
       #MB3_Decoder.OpEnabled := TRUE;
   END_IF;
   IF #_w1 AND NOT "A0302_Bordatrice_RegolazioneFormato".AX_M[4].COut.Standstill AND NOT "A0302_Bordatrice_RegolazioneFormato".AX_M[5].COut.Standstill THEN
       #MB3_Decoder.OpRunning := TRUE;
   END_IF;
   IF #_w1 AND (("A03_HMI".MB3.Button.A0302.Bordatrice.Regolazione.Passaggio_Combo[2].Bwd_Minus AND "A0302_Bordatrice_RegolazioneFormato".AX_M[4].COut.MinusLimitReached AND "A0302_Bordatrice_RegolazioneFormato".AX_M[5].COut.MinusLimitReached) OR ("A03_HMI".MB3.Button.A0302.Bordatrice.Regolazione.Passaggio_Combo[2].Fwd_Plus AND "A0302_Bordatrice_RegolazioneFormato".AX_M[4].COut.PlusLimitReached AND "A0302_Bordatrice_RegolazioneFormato".AX_M[5].COut.PlusLimitReached)) THEN
       #MB3_Decoder.OpDone := TRUE;
   END_IF;
END_REGION

REGION Network 41: MB3 Code 4089 - REGOLAZ. BORDATRICE - PASSAGGIO 02 - COMBO AX-POS
   RUNG wire#powerrail
      { S7_Templates := "SrcType := Int" } EQ_Contact(in1 := #MB3_Decoder.Code, in2 := #"4089_BORDATRICE_PASS02-COMBO_AX-POS")
      wire#w1
      { S7_Templates := "SrcType := LReal" } NE_Contact(in1 := "A0302_Bordatrice_RegolazioneFormato".AX_M[4].COut.ActualPosition, in2 := "A0302_Bordatrice_RegolazioneFormato".HMI.Passaggio02_Combo_TargetPos)
      wire#w2
      Contact( #MB3_Decoder.OperationPlus )
      Coil( "A03_HMI".MB3.Button.A0302.Bordatrice.Regolazione.Passaggio_Combo[2].MoveToPos )
   END_RUNG
   RUNG wire#w1
      { S7_Templates := "SrcType := LReal" } NE_Contact(in1 := "A0302_Bordatrice_RegolazioneFormato".AX_M[5].COut.ActualPosition, in2 := "A0302_Bordatrice_RegolazioneFormato".HMI.Passaggio02_Combo_TargetPos)
   END_RUNG wire#w2
   RUNG wire#w1
      Contact( TRUE )
      S_Coil( #MB3_Decoder.OpEnabled )
   END_RUNG
   RUNG wire#w1
      I_Contact( "A0302_Bordatrice_RegolazioneFormato".AX_M[4].COut.Standstill )
      wire#w3
      S_Coil( #MB3_Decoder.OpRunning )
   END_RUNG
   RUNG wire#w1
      I_Contact( "A0302_Bordatrice_RegolazioneFormato".AX_M[5].COut.Standstill )
   END_RUNG wire#w3
   RUNG wire#w1
      Contact( "A0302_Bordatrice_RegolazioneFormato".AX_M[4].COut.InPosition )
      Contact( "A0302_Bordatrice_RegolazioneFormato".AX_M[5].COut.InPosition )
      S_Coil( #MB3_Decoder.OpDone )
   END_RUNG
   // the same network as SCL:
   #_w1 := #MB3_Decoder.Code = #"4089_BORDATRICE_PASS02-COMBO_AX-POS";
   "A03_HMI".MB3.Button.A0302.Bordatrice.Regolazione.Passaggio_Combo[2].MoveToPos := #_w1 AND (("A0302_Bordatrice_RegolazioneFormato".AX_M[4].COut.ActualPosition <> "A0302_Bordatrice_RegolazioneFormato".HMI.Passaggio02_Combo_TargetPos) OR ("A0302_Bordatrice_RegolazioneFormato".AX_M[5].COut.ActualPosition <> "A0302_Bordatrice_RegolazioneFormato".HMI.Passaggio02_Combo_TargetPos)) AND #MB3_Decoder.OperationPlus;
   IF #_w1 AND TRUE THEN #MB3_Decoder.OpEnabled := TRUE; END_IF;
   IF #_w1 AND (NOT "A0302_Bordatrice_RegolazioneFormato".AX_M[4].COut.Standstill OR NOT "A0302_Bordatrice_RegolazioneFormato".AX_M[5].COut.Standstill) THEN
       #MB3_Decoder.OpRunning := TRUE;
   END_IF;
   IF #_w1 AND "A0302_Bordatrice_RegolazioneFormato".AX_M[4].COut.InPosition AND "A0302_Bordatrice_RegolazioneFormato".AX_M[5].COut.InPosition THEN
       #MB3_Decoder.OpDone := TRUE;
   END_IF;
END_REGION

